LIN {X 0,Y 347.191,Z 710.482,A -85,B 0,C 180,E1 -13656.751,E2 -13656.751} C_VEL
LIN {X 0,Y 346.794,Z 715.502,A -85,B 0,C 180,E1 -13658.78,E2 -13658.78} C_VEL
LIN {X 0,Y 346.624,Z 717.5,A -85,B 0,C 180,E1 -13659.837,E2 -13659.837} C_VEL
LIN {X 0,Y 346.502,Z 719.364,A -85,B 0,C 180,E1 -13661.063,E2 -13661.063} C_VEL
LIN {X 0,Y 346.447,Z 720.875,A -85,B 0,C 180,E1 -13662.443,E2 -13662.443} C_VEL
LIN {X 0,Y 346.474,Z 722.066,A -85,B 0,C 180,E1 -13664.71,E2 -13664.71} C_VEL
LIN {X 0,Y 346.685,Z 721.819,A -85,B 0,C 180,E1 -13666.664,E2 -13666.664} C_VEL
LIN {X 0,Y 346.881,Z 720.668,A -85,B 0,C 180,E1 -13668.31,E2 -13668.31} C_VEL
LIN {X 0,Y 347.167,Z 719.319,A -85,B 0,C 180,E1 -13669.502,E2 -13669.502} C_VEL
LIN {X 0,Y 347.704,Z 716.397,A -85,B 0,C 180,E1 -13671.281,E2 -13671.281} C_VEL
LIN {X 0,Y 348.352,Z 712.378,A -85,B 0,C 180,E1 -13673.047,E2 -13673.047} C_VEL
LIN {X 0,Y 349.156,Z 707.164,A -85,B 0,C 180,E1 -13674.803,E2 -13674.803} C_VEL
LIN {X 0,Y 350.157,Z 700.612,A -85,B 0,C 180,E1 -13676.548,E2 -13676.548} C_VEL
LIN {X 0,Y 351.356,Z 692.175,A -85,B 0,C 180,E1 -13678.338,E2 -13678.338} C_VEL
LIN {X 0,Y 352.806,Z 682.143,A -85,B 0,C 180,E1 -13680,E2 -13680} C_VEL
LIN {X 0,Y 353.932,Z 672.637,A -85,B 0,C 180,E1 -13681.28,E2 -13681.28} C_VEL
LIN {X 0,Y 355.119,Z 662.198,A -85,B 0,C 180,E1 -13682.41,E2 -13682.41} C_VEL
LIN {X 0,Y 356.252,Z 650.75,A -85,B 0,C 180,E1 -13683.393,E2 -13683.393} C_VEL
LIN {X 0,Y 357.17,Z 638.174,A -85,B 0,C 180,E1 -13684.231,E2 -13684.231} C_VEL
LIN {X 0,Y 357.806,Z 624.931,A -85,B 0,C 180,E1 -13684.859,E2 -13684.859} C_VEL
LIN {X 0,Y 358.604,Z 602.211,A -85,B 0,C 180,E1 -13685.518,E2 -13685.518} C_VEL
LIN {X 0,Y 361.1,Z 543.407,A -85,B 0,C 180,E1 -13687.11,E2 -13687.11} C_VEL
LIN {X 0,Y 355.905,Z 531.692,A -85,B 0,C 180,E1 -13688.046,E2 -13688.046} C_VEL
LIN {X 0,Y 350.304,Z 521.591,A -85,B 0,C 180,E1 -13689.037,E2 -13689.037} C_VEL
LIN {X 0,Y 348.516,Z 518.327,A -85,B 0,C 180,E1 -13689.402,E2 -13689.402} C_VEL
LIN {X 0,Y 347.926,Z 516.149,A -85,B 0,C 180,E1 -13690.474,E2 -13690.474} C_VEL
LIN {X 0,Y 347.891,Z 516.152,A -85,B 0,C 180,E1 -13694.15,E2 -13694.15} C_VEL
LIN {X 0,Y 347.883,Z 516.149,A -85,B 0,C 180,E1 -13698.29,E2 -13698.29} C_VEL
LIN {X 0,Y 347.781,Z 516.162,A -85,B 0,C 180,E1 -13701.635,E2 -13701.635} C_VEL
LIN {X 0,Y 347.805,Z 516.16,A -85,B 0,C 180,E1 -13705.109,E2 -13705.109} C_VEL
LIN {X 0,Y 347.806,Z 516.155,A -85,B 0,C 180,E1 -13707.694,E2 -13707.694} C_VEL
LIN {X 0,Y 347.758,Z 516.161,A -85,B 0,C 180,E1 -13710.347,E2 -13710.347} C_VEL
LIN {X 0,Y 347.739,Z 516.164,A -85,B 0,C 180,E1 -13714.464,E2 -13714.464} C_VEL
LIN {X 0,Y 347.769,Z 516.162,A -85,B 0,C 180,E1 -13717.989,E2 -13717.989} C_VEL
LIN {X 0,Y 347.746,Z 516.166,A -85,B 0,C 180,E1 -13721.831,E2 -13721.831} C_VEL
LIN {X 0,Y 347.762,Z 516.169,A -85,B 0,C 180,E1 -13725.017,E2 -13725.017} C_VEL
LIN {X 0,Y 347.747,Z 516.172,A -85,B 0,C 180,E1 -13728.398,E2 -13728.398} C_VEL
LIN {X 0,Y 347.774,Z 516.166,A -85,B 0,C 180,E1 -13732.011,E2 -13732.011} C_VEL
LIN {X 0,Y 347.795,Z 516.377,A -85,B 0,C 180,E1 -13733.619,E2 -13733.619} C_VEL
LIN {X 0,Y 350.137,Z 524.59,A -85,B 0,C 180,E1 -13736.498,E2 -13736.498} C_VEL
LIN {X 0,Y 352.428,Z 533.84,A -85,B 0,C 180,E1 -13739.377,E2 -13739.377} C_VEL
LIN {X 0,Y 354.131,Z 542.797,A -85,B 0,C 180,E1 -13741.88,E2 -13741.88} C_VEL
LIN {X 0,Y 354.087,Z 545.377,A -85,B 0,C 180,E1 -13742.519,E2 -13742.519} C_VEL
LIN {X 0,Y 352.488,Z 556.664,A -85,B 0,C 180,E1 -13745.091,E2 -13745.091} C_VEL
LIN {X 0,Y 356.46,Z 577.198,A -85,B 0,C 180,E1 -13746.185,E2 -13746.185} C_VEL
LIN {X 0,Y 358.79,Z 595.546,A -85,B 0,C 180,E1 -13746.986,E2 -13746.986} C_VEL
LIN {X 0,Y 359.351,Z 604.886,A -85,B 0,C 180,E1 -13747.328,E2 -13747.328} C_VEL
LIN {X 0,Y 356.822,Z 668.886,A -85,B 0,C 180,E1 -13749.047,E2 -13749.047} C_VEL
LIN {X 0,Y 355.901,Z 682.744,A -85,B 0,C 180,E1 -13749.633,E2 -13749.633} C_VEL
LIN {X 0,Y 354.708,Z 694.487,A -85,B 0,C 180,E1 -13750.317,E2 -13750.317} C_VEL
LIN {X 0,Y 353.285,Z 706.996,A -85,B 0,C 180,E1 -13751.29,E2 -13751.29} C_VEL
LIN {X 0,Y 351.842,Z 718.372,A -85,B 0,C 180,E1 -13752.415,E2 -13752.415} C_VEL
LIN {X 0,Y 350.371,Z 732.515,A -85,B 0,C 180,E1 -13753.991,E2 -13753.991} C_VEL
LIN {X 0,Y 349.307,Z 742.889,A -85,B 0,C 180,E1 -13755.434,E2 -13755.434} C_VEL
LIN {X 0,Y 348.389,Z 751.27,A -85,B 0,C 180,E1 -13756.883,E2 -13756.883} C_VEL
LIN {X 0,Y 347.452,Z 759.439,A -85,B 0,C 180,E1 -13758.626,E2 -13758.626} C_VEL
LIN {X 0,Y 346.971,Z 764.991,A -85,B 0,C 180,E1 -13760.086,E2 -13760.086} C_VEL
LIN {X 0,Y 346.551,Z 770.397,A -85,B 0,C 180,E1 -13761.839,E2 -13761.839} C_VEL
LIN {X 0,Y 346.304,Z 774.601,A -85,B 0,C 180,E1 -13763.592,E2 -13763.592} C_VEL
LIN {X 0,Y 346.222,Z 777.723,A -85,B 0,C 180,E1 -13765.343,E2 -13765.343} C_VEL
LIN {X 0,Y 346.186,Z 779.27,A -85,B 0,C 180,E1 -13766.508,E2 -13766.508} C_VEL
LIN {X 0,Y 346.144,Z 780.358,A -85,B 0,C 180,E1 -13767.673,E2 -13767.673} C_VEL
LIN {X 0,Y 346.153,Z 781.038,A -85,B 0,C 180,E1 -13768.837,E2 -13768.837} C_VEL
LIN {X 0,Y 346.173,Z 781.328,A -85,B 0,C 180,E1 -13770,E2 -13770} C_VEL
LIN {X 0,Y 346.137,Z 781.219,A -85,B 0,C 180,E1 -13771.163,E2 -13771.163} C_VEL
LIN {X 0,Y 346.143,Z 780.669,A -85,B 0,C 180,E1 -13772.327,E2 -13772.327} C_VEL
LIN {X 0,Y 346.187,Z 779.723,A -85,B 0,C 180,E1 -13773.492,E2 -13773.492} C_VEL
LIN {X 0,Y 346.224,Z 778.38,A -85,B 0,C 180,E1 -13774.657,E2 -13774.657} C_VEL
LIN {X 0,Y 346.279,Z 776.247,A -85,B 0,C 180,E1 -13776.015,E2 -13776.015} C_VEL
LIN {X 0,Y 346.574,Z 771.638,A -85,B 0,C 180,E1 -13778.16,E2 -13778.16} C_VEL
LIN {X 0,Y 347.014,Z 766.599,A -85,B 0,C 180,E1 -13779.913,E2 -13779.913} C_VEL
LIN {X 0,Y 347.657,Z 760.231,A -85,B 0,C 180,E1 -13781.663,E2 -13781.663} C_VEL
LIN {X 0,Y 348.697,Z 752.269,A -85,B 0,C 180,E1 -13783.402,E2 -13783.402} C_VEL
LIN {X 0,Y 349.658,Z 744.139,A -85,B 0,C 180,E1 -13784.848,E2 -13784.848} C_VEL
LIN {X 0,Y 350.803,Z 734.199,A -85,B 0,C 180,E1 -13786.288,E2 -13786.288} C_VEL
LIN {X 0,Y 352.096,Z 722.923,A -85,B 0,C 180,E1 -13787.571,E2 -13787.571} C_VEL
LIN {X 0,Y 353.243,Z 711.857,A -85,B 0,C 180,E1 -13788.562,E2 -13788.562} C_VEL
LIN {X 0,Y 354.174,Z 700.659,A -85,B 0,C 180,E1 -13789.337,E2 -13789.337} C_VEL
LIN {X 0,Y 355.064,Z 687.97,A -85,B 0,C 180,E1 -13789.964,E2 -13789.964} C_VEL
LIN {X 0,Y 355.672,Z 674.624,A -85,B 0,C 180,E1 -13790.381,E2 -13790.381} C_VEL
LIN {X 0,Y 356.823,Z 601.554,A -85,B 0,C 180,E1 -13791.864,E2 -13791.864} C_VEL
LIN {X 0,Y 352.399,Z 568.881,A -85,B 0,C 180,E1 -13792.872,E2 -13792.872} C_VEL
LIN {X 0,Y 351.1,Z 560.278,A -85,B 0,C 180,E1 -13793.162,E2 -13793.162} C_VEL
LIN {X 0,Y 350.704,Z 555.734,A -85,B 0,C 180,E1 -13793.503,E2 -13793.503} C_VEL
LIN {X 0,Y 352.352,Z 539.207,A -85,B 0,C 180,E1 -13796.985,E2 -13796.985} C_VEL
LIN {X 0,Y 351.415,Z 533.126,A -85,B 0,C 180,E1 -13798.362,E2 -13798.362} C_VEL
LIN {X 0,Y 348.104,Z 517.735,A -85,B 0,C 180,E1 -13802.01,E2 -13802.01} C_VEL
LIN {X 0,Y 347.769,Z 516.167,A -85,B 0,C 180,E1 -13802.426,E2 -13802.426} C_VEL
LIN {X 0,Y 347.768,Z 516.16,A -85,B 0,C 180,E1 -13806.064,E2 -13806.064} C_VEL
LIN {X 0,Y 347.749,Z 516.137,A -85,B 0,C 180,E1 -13808.792,E2 -13808.792} C_VEL
LIN {X 0,Y 347.748,Z 516.169,A -85,B 0,C 180,E1 -13811.829,E2 -13811.829} C_VEL
LIN {X 0,Y 347.765,Z 516.164,A -85,B 0,C 180,E1 -13815.016,E2 -13815.016} C_VEL
LIN {X 0,Y 347.763,Z 516.155,A -85,B 0,C 180,E1 -13818.393,E2 -13818.393} C_VEL
LIN {X 0,Y 347.774,Z 516.16,A -85,B 0,C 180,E1 -13822.01,E2 -13822.01} C_VEL
LIN {X 0,Y 347.739,Z 516.17,A -85,B 0,C 180,E1 -13825.536,E2 -13825.536} C_VEL
LIN {X 0,Y 347.758,Z 516.152,A -85,B 0,C 180,E1 -13829.653,E2 -13829.653} C_VEL
LIN {X 0,Y 347.846,Z 516.155,A -85,B 0,C 180,E1 -13832.744,E2 -13832.744} C_VEL
LIN {X 0,Y 347.777,Z 516.142,A -85,B 0,C 180,E1 -13836.161,E2 -13836.161} C_VEL
LIN {X 0,Y 347.799,Z 516.159,A -85,B 0,C 180,E1 -13839.909,E2 -13839.909} C_VEL
LIN {X 0,Y 347.858,Z 516.14,A -85,B 0,C 180,E1 -13842.359,E2 -13842.359} C_VEL
LIN {X 0,Y 347.89,Z 516.145,A -85,B 0,C 180,E1 -13845.971,E2 -13845.971} C_VEL
LIN {X 0,Y 347.925,Z 516.136,A -85,B 0,C 180,E1 -13849.526,E2 -13849.526} C_VEL
LIN {X 0,Y 348.09,Z 516.108,A -85,B 0,C 180,E1 -13853.042,E2 -13853.042} C_VEL
LIN {X 0,Y 348.201,Z 516.103,A -85,B 0,C 180,E1 -13857.687,E2 -13857.687} C_VEL
LIN {X 0,Y 348.34,Z 516.066,A -85,B 0,C 180,E1 -13860,E2 -13860} C_VEL
LIN {X 0,Y 348.201,Z 516.103,A -85,B 0,C 180,E1 -13862.314,E2 -13862.314} C_VEL
LIN {X 0,Y 348.087,Z 516.11,A -85,B 0,C 180,E1 -13866.958,E2 -13866.958} C_VEL
LIN {X 0,Y 347.921,Z 516.137,A -85,B 0,C 180,E1 -13870.475,E2 -13870.475} C_VEL
LIN {X 0,Y 347.892,Z 516.144,A -85,B 0,C 180,E1 -13874.15,E2 -13874.15} C_VEL
LIN {X 0,Y 347.884,Z 516.144,A -85,B 0,C 180,E1 -13878.291,E2 -13878.291} C_VEL
LIN {X 0,Y 347.782,Z 516.155,A -85,B 0,C 180,E1 -13881.636,E2 -13881.636} C_VEL
LIN {X 0,Y 347.807,Z 516.155,A -85,B 0,C 180,E1 -13885.109,E2 -13885.109} C_VEL
LIN {X 0,Y 347.807,Z 516.156,A -85,B 0,C 180,E1 -13887.695,E2 -13887.695} C_VEL
LIN {X 0,Y 347.766,Z 516.154,A -85,B 0,C 180,E1 -13890.347,E2 -13890.347} C_VEL
LIN {X 0,Y 347.744,Z 516.162,A -85,B 0,C 180,E1 -13894.045,E2 -13894.045} C_VEL
LIN {X 0,Y 347.759,Z 516.17,A -85,B 0,C 180,E1 -13897.322,E2 -13897.322} C_VEL
LIN {X 0,Y 347.73,Z 516.167,A -85,B 0,C 180,E1 -13900.298,E2 -13900.298} C_VEL
LIN {X 0,Y 347.724,Z 516.168,A -85,B 0,C 180,E1 -13903.409,E2 -13903.409} C_VEL
LIN {X 0,Y 347.726,Z 516.169,A -85,B 0,C 180,E1 -13906.687,E2 -13906.687} C_VEL
LIN {X 0,Y 347.747,Z 516.166,A -85,B 0,C 180,E1 -13910.174,E2 -13910.174} C_VEL
LIN {X 0,Y 347.762,Z 516.166,A -85,B 0,C 180,E1 -13912.68,E2 -13912.68} C_VEL
LIN {X 0,Y 347.749,Z 516.164,A -85,B 0,C 180,E1 -13915.957,E2 -13915.957} C_VEL
LIN {X 0,Y 347.77,Z 516.166,A -85,B 0,C 180,E1 -13917.712,E2 -13917.712} C_VEL
LIN {X 0,Y 351.213,Z 530.188,A -85,B 0,C 180,E1 -13920.971,E2 -13920.971} C_VEL
LIN {X 0,Y 352.992,Z 539.619,A -85,B 0,C 180,E1 -13923.039,E2 -13923.039} C_VEL
LIN {X 0,Y 352.487,Z 549.164,A -85,B 0,C 180,E1 -13924.862,E2 -13924.862} C_VEL
LIN {X 0,Y 357.616,Z 575.434,A -85,B 0,C 180,E1 -13925.813,E2 -13925.813} C_VEL
LIN {X 0,Y 357.927,Z 578.608,A -85,B 0,C 180,E1 -13925.902,E2 -13925.902} C_VEL
LIN {X 0,Y 356.197,Z 660.018,A -85,B 0,C 180,E1 -13927.564,E2 -13927.564} C_VEL
LIN {X 0,Y 355.59,Z 672.934,A -85,B 0,C 180,E1 -13928.045,E2 -13928.045} C_VEL
LIN {X 0,Y 354.85,Z 685.894,A -85,B 0,C 180,E1 -13928.789,E2 -13928.789} C_VEL
LIN {X 0,Y 353.861,Z 697.311,A -85,B 0,C 180,E1 -13929.662,E2 -13929.662} C_VEL
LIN {X 0,Y 352.65,Z 708.811,A -85,B 0,C 180,E1 -13930.803,E2 -13930.803} C_VEL
LIN {X 0,Y 351.376,Z 719.111,A -85,B 0,C 180,E1 -13932.091,E2 -13932.091} C_VEL
LIN {X 0,Y 350.306,Z 727.549,A -85,B 0,C 180,E1 -13933.388,E2 -13933.388} C_VEL
LIN {X 0,Y 349.2,Z 736.245,A -85,B 0,C 180,E1 -13935.03,E2 -13935.03} C_VEL
LIN {X 0,Y 348.309,Z 743.998,A -85,B 0,C 180,E1 -13936.88,E2 -13936.88} C_VEL
LIN {X 0,Y 347.34,Z 750.728,A -85,B 0,C 180,E1 -13938.918,E2 -13938.918} C_VEL
LIN {X 0,Y 346.849,Z 755.133,A -85,B 0,C 180,E1 -13940.671,E2 -13940.671} C_VEL
LIN {X 0,Y 346.612,Z 757.443,A -85,B 0,C 180,E1 -13941.84,E2 -13941.84} C_VEL
LIN {X 0,Y 346.328,Z 760.492,A -85,B 0,C 180,E1 -13943.913,E2 -13943.913} C_VEL
LIN {X 0,Y 346.228,Z 761.819,A -85,B 0,C 180,E1 -13945.343,E2 -13945.343} C_VEL
LIN {X 0,Y 346.122,Z 762.712,A -85,B 0,C 180,E1 -13947.673,E2 -13947.673} C_VEL
LIN {X 0,Y 346.132,Z 762.561,A -85,B 0,C 180,E1 -13948.837,E2 -13948.837} C_VEL
LIN {X 0,Y 346.168,Z 761.996,A -85,B 0,C 180,E1 -13950,E2 -13950} C_VEL
LIN {X 0,Y 346.335,Z 759.716,A -85,B 0,C 180,E1 -13952.326,E2 -13952.326} C_VEL
LIN {X 0,Y 346.569,Z 756.887,A -85,B 0,C 180,E1 -13954.07,E2 -13954.07} C_VEL
LIN {X 0,Y 346.939,Z 753.039,A -85,B 0,C 180,E1 -13955.813,E2 -13955.813} C_VEL
LIN {X 0,Y 347.481,Z 747.696,A -85,B 0,C 180,E1 -13957.665,E2 -13957.665} C_VEL
LIN {X 0,Y 348.24,Z 740.577,A -85,B 0,C 180,E1 -13959.584,E2 -13959.584} C_VEL
LIN {X 0,Y 349.222,Z 732.487,A -85,B 0,C 180,E1 -13961.316,E2 -13961.316} C_VEL
LIN {X 0,Y 350.217,Z 724.154,A -85,B 0,C 180,E1 -13962.752,E2 -13962.752} C_VEL
LIN {X 0,Y 351.299,Z 713.922,A -85,B 0,C 180,E1 -13964.186,E2 -13964.186} C_VEL
LIN {X 0,Y 352.354,Z 703.817,A -85,B 0,C 180,E1 -13965.324,E2 -13965.324} C_VEL
LIN {X 0,Y 353.317,Z 692.746,A -85,B 0,C 180,E1 -13966.318,E2 -13966.318} C_VEL
LIN {X 0,Y 354.286,Z 680.233,A -85,B 0,C 180,E1 -13967.162,E2 -13967.162} C_VEL
LIN {X 0,Y 354.855,Z 667.182,A -85,B 0,C 180,E1 -13967.801,E2 -13967.801} C_VEL
LIN {X 0,Y 355.283,Z 653.229,A -85,B 0,C 180,E1 -13968.21,E2 -13968.21} C_VEL
LIN {X 0,Y 356.187,Z 606.958,A -85,B 0,C 180,E1 -13969.133,E2 -13969.133} C_VEL
LIN {X 0,Y 355.84,Z 601.151,A -85,B 0,C 180,E1 -13969.277,E2 -13969.277} C_VEL
LIN {X 0,Y 353.732,Z 591.744,A -85,B 0,C 180,E1 -13969.605,E2 -13969.605} C_VEL
LIN {X 0,Y 351.581,Z 584.287,A -85,B 0,C 180,E1 -13969.899,E2 -13969.899} C_VEL
LIN {X 0,Y 349.907,Z 576.693,A -85,B 0,C 180,E1 -13970.169,E2 -13970.169} C_VEL
LIN {X 0,Y 345.011,Z 549.363,A -85,B 0,C 180,E1 -13971.1,E2 -13971.1} C_VEL
LIN {X 0,Y 345.443,Z 539.348,A -85,B 0,C 180,E1 -13973.024,E2 -13973.024} C_VEL
LIN {X 0,Y 343.402,Z 528.311,A -85,B 0,C 180,E1 -13975.453,E2 -13975.453} C_VEL
LIN {X 0,Y 340.796,Z 517.036,A -85,B 0,C 180,E1 -13978.04,E2 -13978.04} C_VEL
LIN {X 0,Y 340.705,Z 517.046,A -85,B 0,C 180,E1 -13981.043,E2 -13981.043} C_VEL
LIN {X 0,Y 340.718,Z 517.044,A -85,B 0,C 180,E1 -13985.278,E2 -13985.278} C_VEL
LIN {X 0,Y 340.711,Z 517.045,A -85,B 0,C 180,E1 -13988.385,E2 -13988.385} C_VEL
LIN {X 0,Y 340.724,Z 517.039,A -85,B 0,C 180,E1 -13991.303,E2 -13991.303} C_VEL
LIN {X 0,Y 340.719,Z 517.034,A -85,B 0,C 180,E1 -13994.531,E2 -13994.531} C_VEL
LIN {X 0,Y 340.684,Z 517.05,A -85,B 0,C 180,E1 -13998.689,E2 -13998.689} C_VEL
LIN {X 0,Y 340.722,Z 517.043,A -85,B 0,C 180,E1 -14001.814,E2 -14001.814} C_VEL
LIN {X 0,Y 348.431,Z 538.596,A -85,B 0,C 180,E1 -14002.795,E2 -14002.795} C_VEL
LIN {X 0,Y 346.353,Z 619.657,A -85,B 0,C 180,E1 -14004.868,E2 -14004.868} C_VEL
LIN {X 0,Y 345.93,Z 632.4,A -85,B 0,C 180,E1 -14005.417,E2 -14005.417} C_VEL
LIN {X 0,Y 345.376,Z 644.462,A -85,B 0,C 180,E1 -14006.147,E2 -14006.147} C_VEL
LIN {X 0,Y 344.579,Z 656.447,A -85,B 0,C 180,E1 -14007.109,E2 -14007.109} C_VEL
LIN {X 0,Y 343.624,Z 668.932,A -85,B 0,C 180,E1 -14008.392,E2 -14008.392} C_VEL
LIN {X 0,Y 342.759,Z 679.979,A -85,B 0,C 180,E1 -14009.844,E2 -14009.844} C_VEL
LIN {X 0,Y 341.853,Z 689.836,A -85,B 0,C 180,E1 -14011.446,E2 -14011.446} C_VEL
LIN {X 0,Y 341.15,Z 697.81,A -85,B 0,C 180,E1 -14013.049,E2 -14013.049} C_VEL
LIN {X 0,Y 340.546,Z 705.253,A -85,B 0,C 180,E1 -14014.911,E2 -14014.911} C_VEL
LIN {X 0,Y 340.063,Z 711.466,A -85,B 0,C 180,E1 -14016.879,E2 -14016.879} C_VEL
LIN {X 0,Y 339.74,Z 715.579,A -85,B 0,C 180,E1 -14018.57,E2 -14018.57} C_VEL
LIN {X 0,Y 339.45,Z 719.287,A -85,B 0,C 180,E1 -14020.654,E2 -14020.654} C_VEL
LIN {X 0,Y 339.394,Z 721.231,A -85,B 0,C 180,E1 -14022.273,E2 -14022.273} C_VEL
LIN {X 0,Y 339.395,Z 722.535,A -85,B 0,C 180,E1 -14024.383,E2 -14024.383} C_VEL
LIN {X 0,Y 339.607,Z 722.495,A -85,B 0,C 180,E1 -14026.561,E2 -14026.561} C_VEL
LIN {X 0,Y 339.791,Z 721.654,A -85,B 0,C 180,E1 -14028.063,E2 -14028.063} C_VEL
LIN {X 0,Y 340.046,Z 720.452,A -85,B 0,C 180,E1 -14029.28,E2 -14029.28} C_VEL
LIN {X 0,Y 340.615,Z 717.8,A -85,B 0,C 180,E1 -14031.097,E2 -14031.097} C_VEL
LIN {X 0,Y 341.282,Z 714.089,A -85,B 0,C 180,E1 -14032.902,E2 -14032.902} C_VEL
LIN {X 0,Y 342.117,Z 709.218,A -85,B 0,C 180,E1 -14034.696,E2 -14034.696} C_VEL
LIN {X 0,Y 343.1,Z 703.059,A -85,B 0,C 180,E1 -14036.477,E2 -14036.477} C_VEL
LIN {X 0,Y 344.335,Z 695.007,A -85,B 0,C 180,E1 -14038.304,E2 -14038.304} C_VEL
LIN {X 0,Y 345.825,Z 685.582,A -85,B 0,C 180,E1 -14040,E2 -14040} C_VEL
LIN {X 0,Y 347.125,Z 675.585,A -85,B 0,C 180,E1 -14041.45,E2 -14041.45} C_VEL
LIN {X 0,Y 348.546,Z 664.355,A -85,B 0,C 180,E1 -14042.745,E2 -14042.745} C_VEL
LIN {X 0,Y 349.735,Z 653.39,A -85,B 0,C 180,E1 -14043.744,E2 -14043.744} C_VEL
LIN {X 0,Y 350.803,Z 640.159,A -85,B 0,C 180,E1 -14044.668,E2 -14044.668} C_VEL
LIN {X 0,Y 351.489,Z 627.703,A -85,B 0,C 180,E1 -14045.306,E2 -14045.306} C_VEL
LIN {X 0,Y 352.069,Z 611.332,A -85,B 0,C 180,E1 -14045.836,E2 -14045.836} C_VEL
LIN {X 0,Y 355.063,Z 545.537,A -85,B 0,C 180,E1 -14047.672,E2 -14047.672} C_VEL
LIN {X 0,Y 350.562,Z 535.405,A -85,B 0,C 180,E1 -14048.513,E2 -14048.513} C_VEL
LIN {X 0,Y 345.457,Z 526.088,A -85,B 0,C 180,E1 -14049.472,E2 -14049.472} C_VEL
LIN {X 0,Y 341.487,Z 519.336,A -85,B 0,C 180,E1 -14050.246,E2 -14050.246} C_VEL
LIN {X 0,Y 340.844,Z 517.03,A -85,B 0,C 180,E1 -14051.447,E2 -14051.447} C_VEL
LIN {X 0,Y 340.856,Z 517.029,A -85,B 0,C 180,E1 -14054.325,E2 -14054.325} C_VEL
LIN {X 0,Y 340.829,Z 517.028,A -85,B 0,C 180,E1 -14058.466,E2 -14058.466} C_VEL
LIN {X 0,Y 340.747,Z 517.038,A -85,B 0,C 180,E1 -14061.857,E2 -14061.857} C_VEL
LIN {X 0,Y 340.766,Z 517.033,A -85,B 0,C 180,E1 -14065.665,E2 -14065.665} C_VEL
LIN {X 0,Y 340.736,Z 517.036,A -85,B 0,C 180,E1 -14068.32,E2 -14068.32} C_VEL
LIN {X 0,Y 340.698,Z 517.043,A -85,B 0,C 180,E1 -14071.045,E2 -14071.045} C_VEL
LIN {X 0,Y 340.713,Z 517.042,A -85,B 0,C 180,E1 -14075.279,E2 -14075.279} C_VEL
LIN {X 0,Y 340.705,Z 517.042,A -85,B 0,C 180,E1 -14078.387,E2 -14078.387} C_VEL
LIN {X 0,Y 340.694,Z 517.044,A -85,B 0,C 180,E1 -14082.046,E2 -14082.046} C_VEL
LIN {X 0,Y 340.679,Z 517.049,A -85,B 0,C 180,E1 -14085.462,E2 -14085.462} C_VEL
LIN {X 0,Y 340.683,Z 517.05,A -85,B 0,C 180,E1 -14088.691,E2 -14088.691} C_VEL
LIN {X 0,Y 340.741,Z 517.155,A -85,B 0,C 180,E1 -14092.616,E2 -14092.616} C_VEL
LIN {X 0,Y 343.201,Z 525.658,A -85,B 0,C 180,E1 -14095.799,E2 -14095.799} C_VEL
LIN {X 0,Y 345.651,Z 535.486,A -85,B 0,C 180,E1 -14099.011,E2 -14099.011} C_VEL
LIN {X 0,Y 347.353,Z 544.47,A -85,B 0,C 180,E1 -14101.61,E2 -14101.61} C_VEL
LIN {X 0,Y 347.368,Z 547.045,A -85,B 0,C 180,E1 -14102.269,E2 -14102.269} C_VEL
LIN {X 0,Y 345.998,Z 555.843,A -85,B 0,C 180,E1 -14104.328,E2 -14104.328} C_VEL
LIN {X 0,Y 349.88,Z 575.095,A -85,B 0,C 180,E1 -14105.428,E2 -14105.428} C_VEL
LIN {X 0,Y 352.104,Z 591.203,A -85,B 0,C 180,E1 -14106.2,E2 -14106.2} C_VEL
LIN {X 0,Y 353.195,Z 604.961,A -85,B 0,C 180,E1 -14106.761,E2 -14106.761} C_VEL
LIN {X 0,Y 350.497,Z 669.155,A -85,B 0,C 180,E1 -14108.535,E2 -14108.535} C_VEL
LIN {X 0,Y 349.442,Z 683.271,A -85,B 0,C 180,E1 -14109.162,E2 -14109.162} C_VEL
LIN {X 0,Y 348.097,Z 695.544,A -85,B 0,C 180,E1 -14109.927,E2 -14109.927} C_VEL
LIN {X 0,Y 346.613,Z 707.641,A -85,B 0,C 180,E1 -14110.916,E2 -14110.916} C_VEL
LIN {X 0,Y 345.103,Z 718.738,A -85,B 0,C 180,E1 -14112.061,E2 -14112.061} C_VEL
LIN {X 0,Y 343.278,Z 734.494,A -85,B 0,C 180,E1 -14113.956,E2 -14113.956} C_VEL
LIN {X 0,Y 342.177,Z 744.421,A -85,B 0,C 180,E1 -14115.435,E2 -14115.435} C_VEL
LIN {X 0,Y 341.267,Z 752.483,A -85,B 0,C 180,E1 -14116.907,E2 -14116.907} C_VEL
LIN {X 0,Y 340.336,Z 760.405,A -85,B 0,C 180,E1 -14118.687,E2 -14118.687} C_VEL
LIN {X 0,Y 339.759,Z 766.704,A -85,B 0,C 180,E1 -14120.475,E2 -14120.475} C_VEL
LIN {X 0,Y 339.396,Z 771.695,A -85,B 0,C 180,E1 -14122.265,E2 -14122.265} C_VEL
LIN {X 0,Y 339.189,Z 775.535,A -85,B 0,C 180,E1 -14124.054,E2 -14124.054} C_VEL
LIN {X 0,Y 339.123,Z 777.506,A -85,B 0,C 180,E1 -14125.245,E2 -14125.245} C_VEL
LIN {X 0,Y 339.109,Z 779.059,A -85,B 0,C 180,E1 -14126.435,E2 -14126.435} C_VEL
LIN {X 0,Y 339.055,Z 780.156,A -85,B 0,C 180,E1 -14127.624,E2 -14127.624} C_VEL
LIN {X 0,Y 339.054,Z 780.84,A -85,B 0,C 180,E1 -14128.812,E2 -14128.812} C_VEL
LIN {X 0,Y 339.075,Z 781.135,A -85,B 0,C 180,E1 -14130,E2 -14130} C_VEL
LIN {X 0,Y 339.04,Z 781.033,A -85,B 0,C 180,E1 -14131.188,E2 -14131.188} C_VEL
LIN {X 0,Y 339.055,Z 780.49,A -85,B 0,C 180,E1 -14132.376,E2 -14132.376} C_VEL
LIN {X 0,Y 339.11,Z 779.549,A -85,B 0,C 180,E1 -14133.565,E2 -14133.565} C_VEL
LIN {X 0,Y 339.124,Z 778.209,A -85,B 0,C 180,E1 -14134.755,E2 -14134.755} C_VEL
LIN {X 0,Y 339.237,Z 775.369,A -85,B 0,C 180,E1 -14136.542,E2 -14136.542} C_VEL
LIN {X 0,Y 339.531,Z 771.489,A -85,B 0,C 180,E1 -14138.331,E2 -14138.331} C_VEL
LIN {X 0,Y 340.011,Z 766.462,A -85,B 0,C 180,E1 -14140.119,E2 -14140.119} C_VEL
LIN {X 0,Y 340.681,Z 760.114,A -85,B 0,C 180,E1 -14141.905,E2 -14141.905} C_VEL
LIN {X 0,Y 341.779,Z 752.168,A -85,B 0,C 180,E1 -14143.678,E2 -14143.678} C_VEL
LIN {X 0,Y 342.796,Z 744.057,A -85,B 0,C 180,E1 -14145.153,E2 -14145.153} C_VEL
LIN {X 0,Y 343.963,Z 734.146,A -85,B 0,C 180,E1 -14146.621,E2 -14146.621} C_VEL
LIN {X 0,Y 345.18,Z 724.323,A -85,B 0,C 180,E1 -14147.782,E2 -14147.782} C_VEL
LIN {X 0,Y 346.356,Z 713.636,A -85,B 0,C 180,E1 -14148.791,E2 -14148.791} C_VEL
LIN {X 0,Y 347.402,Z 701.87,A -85,B 0,C 180,E1 -14149.653,E2 -14149.653} C_VEL
LIN {X 0,Y 348.342,Z 689.138,A -85,B 0,C 180,E1 -14150.328,E2 -14150.328} C_VEL
LIN {X 0,Y 348.986,Z 676.648,A -85,B 0,C 180,E1 -14150.751,E2 -14150.751} C_VEL
LIN {X 0,Y 350.284,Z 602.378,A -85,B 0,C 180,E1 -14152.293,E2 -14152.293} C_VEL
LIN {X 0,Y 345.913,Z 569.839,A -85,B 0,C 180,E1 -14153.322,E2 -14153.322} C_VEL
LIN {X 0,Y 344.407,Z 560.047,A -85,B 0,C 180,E1 -14153.675,E2 -14153.675} C_VEL
LIN {X 0,Y 343.892,Z 554.129,A -85,B 0,C 180,E1 -14154.125,E2 -14154.125} C_VEL
LIN {X 0,Y 345.334,Z 541.093,A -85,B 0,C 180,E1 -14156.924,E2 -14156.924} C_VEL
LIN {X 0,Y 344.869,Z 536.598,A -85,B 0,C 180,E1 -14157.95,E2 -14157.95} C_VEL
LIN {X 0,Y 341.635,Z 521.206,A -85,B 0,C 180,E1 -14161.639,E2 -14161.639} C_VEL
LIN {X 0,Y 340.735,Z 517.044,A -85,B 0,C 180,E1 -14162.692,E2 -14162.692} C_VEL
LIN {X 0,Y 340.707,Z 517.03,A -85,B 0,C 180,E1 -14166.44,E2 -14166.44} C_VEL
LIN {X 0,Y 340.696,Z 517.029,A -85,B 0,C 180,E1 -14169.752,E2 -14169.752} C_VEL
LIN {X 0,Y 340.672,Z 517.046,A -85,B 0,C 180,E1 -14172.904,E2 -14172.904} C_VEL
LIN {X 0,Y 340.695,Z 517.047,A -85,B 0,C 180,E1 -14176.218,E2 -14176.218} C_VEL
LIN {X 0,Y 340.705,Z 517.045,A -85,B 0,C 180,E1 -14179.748,E2 -14179.748} C_VEL
LIN {X 0,Y 340.702,Z 517.034,A -85,B 0,C 180,E1 -14183.258,E2 -14183.258} C_VEL
LIN {X 0,Y 340.686,Z 517.046,A -85,B 0,C 180,E1 -14186.153,E2 -14186.153} C_VEL
LIN {X 0,Y 340.769,Z 517.025,A -85,B 0,C 180,E1 -14190.332,E2 -14190.332} C_VEL
LIN {X 0,Y 340.798,Z 517.035,A -85,B 0,C 180,E1 -14193.02,E2 -14193.02} C_VEL
LIN {X 0,Y 340.747,Z 517.018,A -85,B 0,C 180,E1 -14195.638,E2 -14195.638} C_VEL
LIN {X 0,Y 340.727,Z 517.042,A -85,B 0,C 180,E1 -14199.473,E2 -14199.473} C_VEL
LIN {X 0,Y 340.85,Z 517.014,A -85,B 0,C 180,E1 -14201.984,E2 -14201.984} C_VEL
LIN {X 0,Y 340.862,Z 517.022,A -85,B 0,C 180,E1 -14205.705,E2 -14205.705} C_VEL
LIN {X 0,Y 340.867,Z 517.017,A -85,B 0,C 180,E1 -14209.306,E2 -14209.306} C_VEL
LIN {X 0,Y 341.057,Z 516.982,A -85,B 0,C 180,E1 -14212.898,E2 -14212.898} C_VEL
LIN {X 0,Y 341.163,Z 516.98,A -85,B 0,C 180,E1 -14217.639,E2 -14217.639} C_VEL
LIN {X 0,Y 341.29,Z 516.943,A -85,B 0,C 180,E1 -14220,E2 -14220} C_VEL
LIN {X 0,Y 341.163,Z 516.979,A -85,B 0,C 180,E1 -14222.362,E2 -14222.362} C_VEL
LIN {X 0,Y 341.054,Z 516.984,A -85,B 0,C 180,E1 -14227.103,E2 -14227.103} C_VEL
LIN {X 0,Y 340.864,Z 517.017,A -85,B 0,C 180,E1 -14230.694,E2 -14230.694} C_VEL
LIN {X 0,Y 340.856,Z 517.021,A -85,B 0,C 180,E1 -14234.325,E2 -14234.325} C_VEL
LIN {X 0,Y 340.83,Z 517.023,A -85,B 0,C 180,E1 -14238.467,E2 -14238.467} C_VEL
LIN {X 0,Y 340.748,Z 517.031,A -85,B 0,C 180,E1 -14241.858,E2 -14241.858} C_VEL
LIN {X 0,Y 340.767,Z 517.036,A -85,B 0,C 180,E1 -14245.665,E2 -14245.665} C_VEL
LIN {X 0,Y 340.737,Z 517.036,A -85,B 0,C 180,E1 -14248.32,E2 -14248.32} C_VEL
LIN {X 0,Y 340.712,Z 517.039,A -85,B 0,C 180,E1 -14251.044,E2 -14251.044} C_VEL
LIN {X 0,Y 340.714,Z 517.036,A -85,B 0,C 180,E1 -14255.28,E2 -14255.28} C_VEL
LIN {X 0,Y 340.707,Z 517.047,A -85,B 0,C 180,E1 -14258.387,E2 -14258.387} C_VEL
LIN {X 0,Y 340.697,Z 517.049,A -85,B 0,C 180,E1 -14262.047,E2 -14262.047} C_VEL
LIN {X 0,Y 340.682,Z 517.05,A -85,B 0,C 180,E1 -14265.463,E2 -14265.463} C_VEL
LIN {X 0,Y 340.685,Z 517.05,A -85,B 0,C 180,E1 -14268.692,E2 -14268.692} C_VEL
LIN {X 0,Y 340.733,Z 517.038,A -85,B 0,C 180,E1 -14271.774,E2 -14271.774} C_VEL
LIN {X 0,Y 340.723,Z 517.035,A -85,B 0,C 180,E1 -14275.596,E2 -14275.596} C_VEL
LIN {X 0,Y 340.724,Z 517.085,A -85,B 0,C 180,E1 -14277.219,E2 -14277.219} C_VEL
LIN {X 0,Y 343.98,Z 530.104,A -85,B 0,C 180,E1 -14280.331,E2 -14280.331} C_VEL
LIN {X 0,Y 346.204,Z 541.28,A -85,B 0,C 180,E1 -14282.824,E2 -14282.824} C_VEL
LIN {X 0,Y 345.792,Z 549.609,A -85,B 0,C 180,E1 -14284.395,E2 -14284.395} C_VEL
LIN {X 0,Y 350.854,Z 575.149,A -85,B 0,C 180,E1 -14285.334,E2 -14285.334} C_VEL
LIN {X 0,Y 351.398,Z 579.233,A -85,B 0,C 180,E1 -14285.462,E2 -14285.462} C_VEL
LIN {X 0,Y 349.649,Z 659.3,A -85,B 0,C 180,E1 -14287.12,E2 -14287.12} C_VEL
LIN {X 0,Y 348.999,Z 672.794,A -85,B 0,C 180,E1 -14287.618,E2 -14287.618} C_VEL
LIN {X 0,Y 348.231,Z 685.556,A -85,B 0,C 180,E1 -14288.354,E2 -14288.354} C_VEL
LIN {X 0,Y 347.178,Z 697.213,A -85,B 0,C 180,E1 -14289.253,E2 -14289.253} C_VEL
LIN {X 0,Y 345.929,Z 708.791,A -85,B 0,C 180,E1 -14290.415,E2 -14290.415} C_VEL
LIN {X 0,Y 344.444,Z 720.168,A -85,B 0,C 180,E1 -14291.871,E2 -14291.871} C_VEL
LIN {X 0,Y 343.247,Z 729.298,A -85,B 0,C 180,E1 -14293.343,E2 -14293.343} C_VEL
LIN {X 0,Y 342.064,Z 738.14,A -85,B 0,C 180,E1 -14295.128,E2 -14295.128} C_VEL
LIN {X 0,Y 341.205,Z 745.193,A -85,B 0,C 180,E1 -14296.905,E2 -14296.905} C_VEL
LIN {X 0,Y 340.338,Z 750.852,A -85,B 0,C 180,E1 -14298.687,E2 -14298.687} C_VEL
LIN {X 0,Y 339.826,Z 755.274,A -85,B 0,C 180,E1 -14300.477,E2 -14300.477} C_VEL
LIN {X 0,Y 339.558,Z 757.592,A -85,B 0,C 180,E1 -14301.67,E2 -14301.67} C_VEL
LIN {X 0,Y 339.247,Z 760.831,A -85,B 0,C 180,E1 -14303.934,E2 -14303.934} C_VEL
LIN {X 0,Y 339.149,Z 761.994,A -85,B 0,C 180,E1 -14305.245,E2 -14305.245} C_VEL
LIN {X 0,Y 339.089,Z 762.636,A -85,B 0,C 180,E1 -14306.435,E2 -14306.435} C_VEL
LIN {X 0,Y 339.034,Z 762.9,A -85,B 0,C 180,E1 -14307.624,E2 -14307.624} C_VEL
LIN {X 0,Y 339.034,Z 762.762,A -85,B 0,C 180,E1 -14308.812,E2 -14308.812} C_VEL
LIN {X 0,Y 339.071,Z 762.202,A -85,B 0,C 180,E1 -14310,E2 -14310} C_VEL
LIN {X 0,Y 339.244,Z 759.935,A -85,B 0,C 180,E1 -14312.375,E2 -14312.375} C_VEL
LIN {X 0,Y 339.495,Z 757.119,A -85,B 0,C 180,E1 -14314.155,E2 -14314.155} C_VEL
LIN {X 0,Y 339.881,Z 753.284,A -85,B 0,C 180,E1 -14315.934,E2 -14315.934} C_VEL
LIN {X 0,Y 340.49,Z 747.453,A -85,B 0,C 180,E1 -14317.979,E2 -14317.979} C_VEL
LIN {X 0,Y 341.251,Z 740.86,A -85,B 0,C 180,E1 -14319.782,E2 -14319.782} C_VEL
LIN {X 0,Y 342.287,Z 732.791,A -85,B 0,C 180,E1 -14321.548,E2 -14321.548} C_VEL
LIN {X 0,Y 343.318,Z 724.488,A -85,B 0,C 180,E1 -14323.013,E2 -14323.013} C_VEL
LIN {X 0,Y 344.449,Z 714.282,A -85,B 0,C 180,E1 -14324.474,E2 -14324.474} C_VEL
LIN {X 0,Y 345.54,Z 704.211,A -85,B 0,C 180,E1 -14325.634,E2 -14325.634} C_VEL
LIN {X 0,Y 346.541,Z 693.205,A -85,B 0,C 180,E1 -14326.646,E2 -14326.646} C_VEL
LIN {X 0,Y 347.528,Z 680.778,A -85,B 0,C 180,E1 -14327.506,E2 -14327.506} C_VEL
LIN {X 0,Y 348.112,Z 668.093,A -85,B 0,C 180,E1 -14328.147,E2 -14328.147} C_VEL
LIN {X 0,Y 348.561,Z 654.621,A -85,B 0,C 180,E1 -14328.567,E2 -14328.567} C_VEL
LIN {X 0,Y 349.948,Z 576.965,A -85,B 0,C 180,E1 -14330.16,E2 -14330.16} C_VEL
LIN {X 0,Y 349.907,Z 576.693,A -85,B 0,C 180,E1 -14330.169,E2 -14330.169} C_VEL
LIN {X 0,Y 348.704,Z 573.037,A -85,B 0,C 180,E1 -14330.326,E2 -14330.326} C_VEL
LIN {X 0,Y 345.131,Z 567.751,A -85,B 0,C 180,E1 -14330.676,E2 -14330.676} C_VEL
LIN {X 0,Y 341.444,Z 562.504,A -85,B 0,C 180,E1 -14331.042,E2 -14331.042} C_VEL
LIN {X 0,Y 340.067,Z 558.89,A -85,B 0,C 180,E1 -14331.218,E2 -14331.218} C_VEL
LIN {X 0,Y 338.228,Z 549.527,A -85,B 0,C 180,E1 -14331.559,E2 -14331.559} C_VEL
LIN {X 0,Y 338.635,Z 540.949,A -85,B 0,C 180,E1 -14333.223,E2 -14333.223} C_VEL
LIN {X 0,Y 336.508,Z 529.712,A -85,B 0,C 180,E1 -14335.735,E2 -14335.735} C_VEL
LIN {X 0,Y 333.758,Z 517.913,A -85,B 0,C 180,E1 -14338.511,E2 -14338.511} C_VEL
LIN {X 0,Y 333.634,Z 517.929,A -85,B 0,C 180,E1 -14341.777,E2 -14341.777} C_VEL
LIN {X 0,Y 333.686,Z 517.92,A -85,B 0,C 180,E1 -14344.773,E2 -14344.773} C_VEL
LIN {X 0,Y 333.678,Z 517.922,A -85,B 0,C 180,E1 -14348.802,E2 -14348.802} C_VEL
LIN {X 0,Y 333.687,Z 517.92,A -85,B 0,C 180,E1 -14352.509,E2 -14352.509} C_VEL
LIN {X 0,Y 333.632,Z 517.916,A -85,B 0,C 180,E1 -14355.96,E2 -14355.96} C_VEL
LIN {X 0,Y 333.645,Z 517.925,A -85,B 0,C 180,E1 -14359.314,E2 -14359.314} C_VEL
LIN {X 0,Y 333.676,Z 517.922,A -85,B 0,C 180,E1 -14361.459,E2 -14361.459} C_VEL
LIN {X 0,Y 341.579,Z 540.099,A -85,B 0,C 180,E1 -14362.499,E2 -14362.499} C_VEL
LIN {X 0,Y 339.45,Z 620.15,A -85,B 0,C 180,E1 -14364.615,E2 -14364.615} C_VEL
LIN {X 0,Y 338.957,Z 634.061,A -85,B 0,C 180,E1 -14365.236,E2 -14365.236} C_VEL
LIN {X 0,Y 338.338,Z 646.332,A -85,B 0,C 180,E1 -14366.022,E2 -14366.022} C_VEL
LIN {X 0,Y 337.491,Z 658.633,A -85,B 0,C 180,E1 -14367.059,E2 -14367.059} C_VEL
LIN {X 0,Y 336.641,Z 669.245,A -85,B 0,C 180,E1 -14368.187,E2 -14368.187} C_VEL
LIN {X 0,Y 335.798,Z 679.738,A -85,B 0,C 180,E1 -14369.576,E2 -14369.576} C_VEL
LIN {X 0,Y 334.898,Z 689.333,A -85,B 0,C 180,E1 -14371.14,E2 -14371.14} C_VEL
LIN {X 0,Y 334.187,Z 697.547,A -85,B 0,C 180,E1 -14372.78,E2 -14372.78} C_VEL
LIN {X 0,Y 333.578,Z 704.465,A -85,B 0,C 180,E1 -14374.478,E2 -14374.478} C_VEL
LIN {X 0,Y 333.095,Z 710.602,A -85,B 0,C 180,E1 -14376.366,E2 -14376.366} C_VEL
LIN {X 0,Y 332.699,Z 715.604,A -85,B 0,C 180,E1 -14378.348,E2 -14378.348} C_VEL
LIN {X 0,Y 332.413,Z 719.122,A -85,B 0,C 180,E1 -14380.228,E2 -14380.228} C_VEL
LIN {X 0,Y 332.322,Z 721.539,A -85,B 0,C 180,E1 -14382.109,E2 -14382.109} C_VEL
LIN {X 0,Y 332.302,Z 722.944,A -85,B 0,C 180,E1 -14384.041,E2 -14384.041} C_VEL
LIN {X 0,Y 332.371,Z 723.288,A -85,B 0,C 180,E1 -14385.301,E2 -14385.301} C_VEL
LIN {X 0,Y 332.549,Z 723.143,A -85,B 0,C 180,E1 -14386.557,E2 -14386.557} C_VEL
LIN {X 0,Y 332.696,Z 722.587,A -85,B 0,C 180,E1 -14387.804,E2 -14387.804} C_VEL
LIN {X 0,Y 332.949,Z 721.593,A -85,B 0,C 180,E1 -14389.048,E2 -14389.048} C_VEL
LIN {X 0,Y 333.29,Z 720.104,A -85,B 0,C 180,E1 -14390.288,E2 -14390.288} C_VEL
LIN {X 0,Y 333.875,Z 717.307,A -85,B 0,C 180,E1 -14391.999,E2 -14391.999} C_VEL
LIN {X 0,Y 334.712,Z 712.853,A -85,B 0,C 180,E1 -14393.973,E2 -14393.973} C_VEL
LIN {X 0,Y 335.692,Z 707.452,A -85,B 0,C 180,E1 -14395.798,E2 -14395.798} C_VEL
LIN {X 0,Y 336.898,Z 700.686,A -85,B 0,C 180,E1 -14397.609,E2 -14397.609} C_VEL
LIN {X 0,Y 338.038,Z 693.717,A -85,B 0,C 180,E1 -14399.122,E2 -14399.122} C_VEL
LIN {X 0,Y 339.403,Z 685.421,A -85,B 0,C 180,E1 -14400.593,E2 -14400.593} C_VEL
LIN {X 0,Y 340.803,Z 675.22,A -85,B 0,C 180,E1 -14402.068,E2 -14402.068} C_VEL
LIN {X 0,Y 342.306,Z 663.738,A -85,B 0,C 180,E1 -14403.384,E2 -14403.384} C_VEL
LIN {X 0,Y 343.581,Z 652.345,A -85,B 0,C 180,E1 -14404.399,E2 -14404.399} C_VEL
LIN {X 0,Y 344.613,Z 639.994,A -85,B 0,C 180,E1 -14405.265,E2 -14405.265} C_VEL
LIN {X 0,Y 345.344,Z 627.265,A -85,B 0,C 180,E1 -14405.913,E2 -14405.913} C_VEL
LIN {X 0,Y 346.16,Z 608.114,A -85,B 0,C 180,E1 -14406.521,E2 -14406.521} C_VEL
LIN {X 0,Y 349.053,Z 547.672,A -85,B 0,C 180,E1 -14408.255,E2 -14408.255} C_VEL
LIN {X 0,Y 345.232,Z 539.034,A -85,B 0,C 180,E1 -14409.022,E2 -14409.022} C_VEL
LIN {X 0,Y 340.523,Z 530.408,A -85,B 0,C 180,E1 -14409.936,E2 -14409.936} C_VEL
LIN {X 0,Y 336.263,Z 523.502,A -85,B 0,C 180,E1 -14410.799,E2 -14410.799} C_VEL
LIN {X 0,Y 334.452,Z 520.265,A -85,B 0,C 180,E1 -14411.208,E2 -14411.208} C_VEL
LIN {X 0,Y 333.784,Z 517.908,A -85,B 0,C 180,E1 -14412.463,E2 -14412.463} C_VEL
LIN {X 0,Y 333.77,Z 517.911,A -85,B 0,C 180,E1 -14415.886,E2 -14415.886} C_VEL
LIN {X 0,Y 333.789,Z 517.906,A -85,B 0,C 180,E1 -14418.655,E2 -14418.655} C_VEL
LIN {X 0,Y 333.685,Z 517.919,A -85,B 0,C 180,E1 -14422.278,E2 -14422.278} C_VEL
LIN {X 0,Y 333.729,Z 517.911,A -85,B 0,C 180,E1 -14426.247,E2 -14426.247} C_VEL
LIN {X 0,Y 333.705,Z 517.914,A -85,B 0,C 180,E1 -14428.972,E2 -14428.972} C_VEL
LIN {X 0,Y 333.638,Z 517.921,A -85,B 0,C 180,E1 -14432.587,E2 -14432.587} C_VEL
LIN {X 0,Y 333.671,Z 517.916,A -85,B 0,C 180,E1 -14436.14,E2 -14436.14} C_VEL
LIN {X 0,Y 333.642,Z 517.927,A -85,B 0,C 180,E1 -14439.193,E2 -14439.193} C_VEL
LIN {X 0,Y 333.628,Z 517.926,A -85,B 0,C 180,E1 -14442.501,E2 -14442.501} C_VEL
LIN {X 0,Y 333.617,Z 517.929,A -85,B 0,C 180,E1 -14445.96,E2 -14445.96} C_VEL
LIN {X 0,Y 333.644,Z 517.927,A -85,B 0,C 180,E1 -14449.316,E2 -14449.316} C_VEL
LIN {X 0,Y 333.669,Z 518.007,A -85,B 0,C 180,E1 -14451.516,E2 -14451.516} C_VEL
LIN {X 0,Y 335.971,Z 525.722,A -85,B 0,C 180,E1 -14454.669,E2 -14454.669} C_VEL
LIN {X 0,Y 338.133,Z 534.074,A -85,B 0,C 180,E1 -14457.606,E2 -14457.606} C_VEL
LIN {X 0,Y 340.175,Z 543.502,A -85,B 0,C 180,E1 -14460.542,E2 -14460.542} C_VEL
LIN {X 0,Y 340.781,Z 547.49,A -85,B 0,C 180,E1 -14461.685,E2 -14461.685} C_VEL
LIN {X 0,Y 339.617,Z 555.073,A -85,B 0,C 180,E1 -14463.521,E2 -14463.521} C_VEL
LIN {X 0,Y 343.128,Z 572.133,A -85,B 0,C 180,E1 -14464.569,E2 -14464.569} C_VEL
LIN {X 0,Y 345.411,Z 586.562,A -85,B 0,C 180,E1 -14465.34,E2 -14465.34} C_VEL
LIN {X 0,Y 347.021,Z 603.168,A -85,B 0,C 180,E1 -14466.076,E2 -14466.076} C_VEL
LIN {X 0,Y 346.943,Z 609.244,A -85,B 0,C 180,E1 -14466.269,E2 -14466.269} C_VEL
LIN {X 0,Y 344.259,Z 668.434,A -85,B 0,C 180,E1 -14467.969,E2 -14467.969} C_VEL
LIN {X 0,Y 343.113,Z 682.555,A -85,B 0,C 180,E1 -14468.602,E2 -14468.602} C_VEL
LIN {X 0,Y 341.725,Z 694.829,A -85,B 0,C 180,E1 -14469.379,E2 -14469.379} C_VEL
LIN {X 0,Y 340.162,Z 706.941,A -85,B 0,C 180,E1 -14470.383,E2 -14470.383} C_VEL
LIN {X 0,Y 338.593,Z 718.011,A -85,B 0,C 180,E1 -14471.547,E2 -14471.547} C_VEL
LIN {X 0,Y 335.913,Z 738.418,A -85,B 0,C 180,E1 -14474.218,E2 -14474.218} C_VEL
LIN {X 0,Y 334.838,Z 747.532,A -85,B 0,C 180,E1 -14475.723,E2 -14475.723} C_VEL
LIN {X 0,Y 333.802,Z 756.399,A -85,B 0,C 180,E1 -14477.537,E2 -14477.537} C_VEL
LIN {X 0,Y 333.031,Z 763.486,A -85,B 0,C 180,E1 -14479.359,E2 -14479.359} C_VEL
LIN {X 0,Y 332.449,Z 769.923,A -85,B 0,C 180,E1 -14481.49,E2 -14481.49} C_VEL
LIN {X 0,Y 332.157,Z 774.147,A -85,B 0,C 180,E1 -14483.317,E2 -14483.317} C_VEL
LIN {X 0,Y 332.028,Z 777.289,A -85,B 0,C 180,E1 -14485.143,E2 -14485.143} C_VEL
LIN {X 0,Y 332.033,Z 778.848,A -85,B 0,C 180,E1 -14486.359,E2 -14486.359} C_VEL
LIN {X 0,Y 331.97,Z 779.954,A -85,B 0,C 180,E1 -14487.573,E2 -14487.573} C_VEL
LIN {X 0,Y 331.958,Z 780.642,A -85,B 0,C 180,E1 -14488.787,E2 -14488.787} C_VEL
LIN {X 0,Y 331.978,Z 780.942,A -85,B 0,C 180,E1 -14490,E2 -14490} C_VEL
LIN {X 0,Y 331.945,Z 780.846,A -85,B 0,C 180,E1 -14491.213,E2 -14491.213} C_VEL
LIN {X 0,Y 331.969,Z 780.311,A -85,B 0,C 180,E1 -14492.427,E2 -14492.427} C_VEL
LIN {X 0,Y 332.034,Z 779.374,A -85,B 0,C 180,E1 -14493.641,E2 -14493.641} C_VEL
LIN {X 0,Y 332.086,Z 776.529,A -85,B 0,C 180,E1 -14495.917,E2 -14495.917} C_VEL
LIN {X 0,Y 332.362,Z 772.764,A -85,B 0,C 180,E1 -14497.9,E2 -14497.9} C_VEL
LIN {X 0,Y 332.783,Z 768.135,A -85,B 0,C 180,E1 -14499.727,E2 -14499.727} C_VEL
LIN {X 0,Y 333.561,Z 761.13,A -85,B 0,C 180,E1 -14501.854,E2 -14501.854} C_VEL
LIN {X 0,Y 334.656,Z 753.54,A -85,B 0,C 180,E1 -14503.665,E2 -14503.665} C_VEL
LIN {X 0,Y 335.945,Z 743.977,A -85,B 0,C 180,E1 -14505.469,E2 -14505.469} C_VEL
LIN {X 0,Y 337.145,Z 734.092,A -85,B 0,C 180,E1 -14506.968,E2 -14506.968} C_VEL
LIN {X 0,Y 338.589,Z 722.9,A -85,B 0,C 180,E1 -14508.297,E2 -14508.297} C_VEL
LIN {X 0,Y 339.828,Z 711.925,A -85,B 0,C 180,E1 -14509.323,E2 -14509.323} C_VEL
LIN {X 0,Y 340.975,Z 699.715,A -85,B 0,C 180,E1 -14510.196,E2 -14510.196} C_VEL
LIN {X 0,Y 341.824,Z 686.75,A -85,B 0,C 180,E1 -14510.851,E2 -14510.851} C_VEL
LIN {X 0,Y 342.489,Z 674.346,A -85,B 0,C 180,E1 -14511.242,E2 -14511.242} C_VEL
LIN {X 0,Y 343.772,Z 603.154,A -85,B 0,C 180,E1 -14512.739,E2 -14512.739} C_VEL
LIN {X 0,Y 338.835,Z 566.34,A -85,B 0,C 180,E1 -14513.938,E2 -14513.938} C_VEL
LIN {X 0,Y 337.728,Z 559.865,A -85,B 0,C 180,E1 -14514.195,E2 -14514.195} C_VEL
LIN {X 0,Y 337.204,Z 552.373,A -85,B 0,C 180,E1 -14514.799,E2 -14514.799} C_VEL
LIN {X 0,Y 338.372,Z 541.515,A -85,B 0,C 180,E1 -14517.189,E2 -14517.189} C_VEL
LIN {X 0,Y 337.179,Z 534.256,A -85,B 0,C 180,E1 -14518.904,E2 -14518.904} C_VEL
LIN {X 0,Y 333.688,Z 517.922,A -85,B 0,C 180,E1 -14522.962,E2 -14522.962} C_VEL
LIN {X 0,Y 333.662,Z 517.899,A -85,B 0,C 180,E1 -14526.832,E2 -14526.832} C_VEL
LIN {X 0,Y 333.644,Z 517.921,A -85,B 0,C 180,E1 -14530.767,E2 -14530.767} C_VEL
LIN {X 0,Y 333.621,Z 517.921,A -85,B 0,C 180,E1 -14534.255,E2 -14534.255} C_VEL
LIN {X 0,Y 333.676,Z 517.911,A -85,B 0,C 180,E1 -14537.624,E2 -14537.624} C_VEL
LIN {X 0,Y 333.673,Z 517.922,A -85,B 0,C 180,E1 -14541.196,E2 -14541.196} C_VEL
LIN {X 0,Y 333.68,Z 517.918,A -85,B 0,C 180,E1 -14545.225,E2 -14545.225} C_VEL
LIN {X 0,Y 333.691,Z 517.903,A -85,B 0,C 180,E1 -14549.637,E2 -14549.637} C_VEL
LIN {X 0,Y 333.738,Z 517.911,A -85,B 0,C 180,E1 -14552.401,E2 -14552.401} C_VEL
LIN {X 0,Y 333.719,Z 517.897,A -85,B 0,C 180,E1 -14555.09,E2 -14555.09} C_VEL
LIN {X 0,Y 333.666,Z 517.92,A -85,B 0,C 180,E1 -14559.018,E2 -14559.018} C_VEL
LIN {X 0,Y 333.786,Z 517.896,A -85,B 0,C 180,E1 -14561.589,E2 -14561.589} C_VEL
LIN {X 0,Y 333.801,Z 517.898,A -85,B 0,C 180,E1 -14565.577,E2 -14565.577} C_VEL
LIN {X 0,Y 333.83,Z 517.896,A -85,B 0,C 180,E1 -14569.078,E2 -14569.078} C_VEL
LIN {X 0,Y 334.009,Z 517.858,A -85,B 0,C 180,E1 -14572.747,E2 -14572.747} C_VEL
LIN {X 0,Y 333.808,Z 517.905,A -85,B 0,C 180,E1 -14575.169,E2 -14575.169} C_VEL
LIN {X 0,Y 334.1,Z 517.86,A -85,B 0,C 180,E1 -14577.589,E2 -14577.589} C_VEL
LIN {X 0,Y 334.241,Z 517.821,A -85,B 0,C 180,E1 -14580,E2 -14580} C_VEL
LIN {X 0,Y 334.101,Z 517.859,A -85,B 0,C 180,E1 -14582.411,E2 -14582.411} C_VEL
LIN {X 0,Y 333.988,Z 517.867,A -85,B 0,C 180,E1 -14586.596,E2 -14586.596} C_VEL
LIN {X 0,Y 333.844,Z 517.885,A -85,B 0,C 180,E1 -14589.696,E2 -14589.696} C_VEL
LIN {X 0,Y 333.79,Z 517.903,A -85,B 0,C 180,E1 -14593.392,E2 -14593.392} C_VEL
LIN {X 0,Y 333.739,Z 517.894,A -85,B 0,C 180,E1 -14597.147,E2 -14597.147} C_VEL
LIN {X 0,Y 333.73,Z 517.913,A -85,B 0,C 180,E1 -14599.691,E2 -14599.691} C_VEL
LIN {X 0,Y 333.687,Z 517.909,A -85,B 0,C 180,E1 -14602.279,E2 -14602.279} C_VEL
LIN {X 0,Y 333.731,Z 517.912,A -85,B 0,C 180,E1 -14606.247,E2 -14606.247} C_VEL
LIN {X 0,Y 333.707,Z 517.904,A -85,B 0,C 180,E1 -14608.973,E2 -14608.973} C_VEL
LIN {X 0,Y 333.647,Z 517.925,A -85,B 0,C 180,E1 -14612.59,E2 -14612.59} C_VEL
LIN {X 0,Y 333.673,Z 517.919,A -85,B 0,C 180,E1 -14616.14,E2 -14616.14} C_VEL
LIN {X 0,Y 333.644,Z 517.92,A -85,B 0,C 180,E1 -14619.193,E2 -14619.193} C_VEL
LIN {X 0,Y 333.631,Z 517.93,A -85,B 0,C 180,E1 -14622.501,E2 -14622.501} C_VEL
LIN {X 0,Y 333.62,Z 517.928,A -85,B 0,C 180,E1 -14625.96,E2 -14625.96} C_VEL
LIN {X 0,Y 333.646,Z 517.921,A -85,B 0,C 180,E1 -14629.316,E2 -14629.316} C_VEL
LIN {X 0,Y 333.665,Z 517.925,A -85,B 0,C 180,E1 -14633.169,E2 -14633.169} C_VEL
LIN {X 0,Y 333.681,Z 517.991,A -85,B 0,C 180,E1 -14636.73,E2 -14636.73} C_VEL
LIN {X 0,Y 336.743,Z 529.983,A -85,B 0,C 180,E1 -14639.648,E2 -14639.648} C_VEL
LIN {X 0,Y 339.143,Z 541.185,A -85,B 0,C 180,E1 -14642.209,E2 -14642.209} C_VEL
LIN {X 0,Y 339.428,Z 544.555,A -85,B 0,C 180,E1 -14642.916,E2 -14642.916} C_VEL
LIN {X 0,Y 339.139,Z 549.814,A -85,B 0,C 180,E1 -14643.885,E2 -14643.885} C_VEL
LIN {X 0,Y 344.419,Z 576.436,A -85,B 0,C 180,E1 -14644.894,E2 -14644.894} C_VEL
LIN {X 0,Y 344.875,Z 580.444,A -85,B 0,C 180,E1 -14645.018,E2 -14645.018} C_VEL
LIN {X 0,Y 343.069,Z 659.892,A -85,B 0,C 180,E1 -14646.695,E2 -14646.695} C_VEL
LIN {X 0,Y 342.371,Z 673.222,A -85,B 0,C 180,E1 -14647.201,E2 -14647.201} C_VEL
LIN {X 0,Y 341.557,Z 686.37,A -85,B 0,C 180,E1 -14647.983,E2 -14647.983} C_VEL
LIN {X 0,Y 340.387,Z 698.777,A -85,B 0,C 180,E1 -14648.978,E2 -14648.978} C_VEL
LIN {X 0,Y 339.08,Z 710.023,A -85,B 0,C 180,E1 -14650.16,E2 -14650.16} C_VEL
LIN {X 0,Y 337.696,Z 720.186,A -85,B 0,C 180,E1 -14651.496,E2 -14651.496} C_VEL
LIN {X 0,Y 336.41,Z 729.357,A -85,B 0,C 180,E1 -14652.994,E2 -14652.994} C_VEL
LIN {X 0,Y 335.27,Z 737.456,A -85,B 0,C 180,E1 -14654.638,E2 -14654.638} C_VEL
LIN {X 0,Y 334.256,Z 745.295,A -85,B 0,C 180,E1 -14656.628,E2 -14656.628} C_VEL
LIN {X 0,Y 333.351,Z 750.976,A -85,B 0,C 180,E1 -14658.447,E2 -14658.447} C_VEL
LIN {X 0,Y 332.785,Z 755.415,A -85,B 0,C 180,E1 -14660.273,E2 -14660.273} C_VEL
LIN {X 0,Y 332.523,Z 757.741,A -85,B 0,C 180,E1 -14661.492,E2 -14661.492} C_VEL
LIN {X 0,Y 332.282,Z 759.643,A -85,B 0,C 180,E1 -14662.709,E2 -14662.709} C_VEL
LIN {X 0,Y 332.14,Z 761.203,A -85,B 0,C 180,E1 -14663.999,E2 -14663.999} C_VEL
LIN {X 0,Y 332.017,Z 762.818,A -85,B 0,C 180,E1 -14666.359,E2 -14666.359} C_VEL
LIN {X 0,Y 331.949,Z 763.087,A -85,B 0,C 180,E1 -14667.573,E2 -14667.573} C_VEL
LIN {X 0,Y 331.939,Z 762.961,A -85,B 0,C 180,E1 -14668.787,E2 -14668.787} C_VEL
LIN {X 0,Y 331.974,Z 762.409,A -85,B 0,C 180,E1 -14670,E2 -14670} C_VEL
LIN {X 0,Y 332.154,Z 760.155,A -85,B 0,C 180,E1 -14672.425,E2 -14672.425} C_VEL
LIN {X 0,Y 332.426,Z 757.35,A -85,B 0,C 180,E1 -14674.243,E2 -14674.243} C_VEL
LIN {X 0,Y 332.827,Z 753.529,A -85,B 0,C 180,E1 -14676.06,E2 -14676.06} C_VEL
LIN {X 0,Y 333.432,Z 747.963,A -85,B 0,C 180,E1 -14678.073,E2 -14678.073} C_VEL
LIN {X 0,Y 334.263,Z 741.143,A -85,B 0,C 180,E1 -14679.989,E2 -14679.989} C_VEL
LIN {X 0,Y 335.361,Z 733.092,A -85,B 0,C 180,E1 -14681.79,E2 -14681.79} C_VEL
LIN {X 0,Y 336.431,Z 724.82,A -85,B 0,C 180,E1 -14683.284,E2 -14683.284} C_VEL
LIN {X 0,Y 337.604,Z 714.641,A -85,B 0,C 180,E1 -14684.774,E2 -14684.774} C_VEL
LIN {X 0,Y 338.739,Z 704.603,A -85,B 0,C 180,E1 -14685.956,E2 -14685.956} C_VEL
LIN {X 0,Y 339.775,Z 693.654,A -85,B 0,C 180,E1 -14686.987,E2 -14686.987} C_VEL
LIN {X 0,Y 340.798,Z 681.32,A -85,B 0,C 180,E1 -14687.863,E2 -14687.863} C_VEL
LIN {X 0,Y 341.406,Z 668.582,A -85,B 0,C 180,E1 -14688.525,E2 -14688.525} C_VEL
LIN {X 0,Y 341.884,Z 655.907,A -85,B 0,C 180,E1 -14688.939,E2 -14688.939} C_VEL
LIN {X 0,Y 343.383,Z 578.072,A -85,B 0,C 180,E1 -14690.564,E2 -14690.564} C_VEL
LIN {X 0,Y 340.067,Z 558.89,A -85,B 0,C 180,E1 -14691.218,E2 -14691.218} C_VEL
LIN {X 0,Y 338.722,Z 555.273,A -85,B 0,C 180,E1 -14691.425,E2 -14691.425} C_VEL
LIN {X 0,Y 336.744,Z 552.17,A -85,B 0,C 180,E1 -14691.733,E2 -14691.733} C_VEL
LIN {X 0,Y 333.395,Z 547.706,A -85,B 0,C 180,E1 -14692.42,E2 -14692.42} C_VEL
LIN {X 0,Y 331.962,Z 544.7,A -85,B 0,C 180,E1 -14693.006,E2 -14693.006} C_VEL
LIN {X 0,Y 331.826,Z 543.387,A -85,B 0,C 180,E1 -14693.273,E2 -14693.273} C_VEL
LIN {X 0,Y 330.696,Z 536.16,A -85,B 0,C 180,E1 -14694.851,E2 -14694.851} C_VEL
LIN {X 0,Y 328.291,Z 525.22,A -85,B 0,C 180,E1 -14697.404,E2 -14697.404} C_VEL
LIN {X 0,Y 326.694,Z 518.791,A -85,B 0,C 180,E1 -14698.947,E2 -14698.947} C_VEL
LIN {X 0,Y 326.618,Z 518.8,A -85,B 0,C 180,E1 -14702.945,E2 -14702.945} C_VEL
LIN {X 0,Y 326.613,Z 518.8,A -85,B 0,C 180,E1 -14705.519,E2 -14705.519} C_VEL
LIN {X 0,Y 326.642,Z 518.793,A -85,B 0,C 180,E1 -14709.233,E2 -14709.233} C_VEL
LIN {X 0,Y 326.625,Z 518.8,A -85,B 0,C 180,E1 -14712.98,E2 -14712.98} C_VEL
LIN {X 0,Y 326.584,Z 518.802,A -85,B 0,C 180,E1 -14717.025,E2 -14717.025} C_VEL
LIN {X 0,Y 326.617,Z 518.807,A -85,B 0,C 180,E1 -14721.124,E2 -14721.124} C_VEL
LIN {X 0,Y 334.674,Z 541.446,A -85,B 0,C 180,E1 -14722.202,E2 -14722.202} C_VEL
LIN {X 0,Y 332.561,Z 620.658,A -85,B 0,C 180,E1 -14724.351,E2 -14724.351} C_VEL
LIN {X 0,Y 332.062,Z 634.129,A -85,B 0,C 180,E1 -14724.963,E2 -14724.963} C_VEL
LIN {X 0,Y 331.363,Z 647.081,A -85,B 0,C 180,E1 -14725.807,E2 -14725.807} C_VEL
LIN {X 0,Y 330.547,Z 658.707,A -85,B 0,C 180,E1 -14726.805,E2 -14726.805} C_VEL
LIN {X 0,Y 329.641,Z 670.123,A -85,B 0,C 180,E1 -14728.041,E2 -14728.041} C_VEL
LIN {X 0,Y 328.782,Z 680.747,A -85,B 0,C 180,E1 -14729.49,E2 -14729.49} C_VEL
LIN {X 0,Y 327.827,Z 690.374,A -85,B 0,C 180,E1 -14731.103,E2 -14731.103} C_VEL
LIN {X 0,Y 327.074,Z 698.734,A -85,B 0,C 180,E1 -14732.831,E2 -14732.831} C_VEL
LIN {X 0,Y 326.43,Z 706.058,A -85,B 0,C 180,E1 -14734.72,E2 -14734.72} C_VEL
LIN {X 0,Y 325.984,Z 711.58,A -85,B 0,C 180,E1 -14736.493,E2 -14736.493} C_VEL
LIN {X 0,Y 325.597,Z 716.396,A -85,B 0,C 180,E1 -14738.472,E2 -14738.472} C_VEL
LIN {X 0,Y 325.389,Z 718.885,A -85,B 0,C 180,E1 -14739.782,E2 -14739.782} C_VEL
LIN {X 0,Y 325.244,Z 721.832,A -85,B 0,C 180,E1 -14741.942,E2 -14741.942} C_VEL
LIN {X 0,Y 325.207,Z 723.27,A -85,B 0,C 180,E1 -14743.683,E2 -14743.683} C_VEL
LIN {X 0,Y 325.262,Z 723.781,A -85,B 0,C 180,E1 -14744.972,E2 -14744.972} C_VEL
LIN {X 0,Y 325.437,Z 723.854,A -85,B 0,C 180,E1 -14746.356,E2 -14746.356} C_VEL
LIN {X 0,Y 325.595,Z 723.465,A -85,B 0,C 180,E1 -14747.534,E2 -14747.534} C_VEL
LIN {X 0,Y 325.842,Z 722.621,A -85,B 0,C 180,E1 -14748.806,E2 -14748.806} C_VEL
LIN {X 0,Y 326.191,Z 721.352,A -85,B 0,C 180,E1 -14750.074,E2 -14750.074} C_VEL
LIN {X 0,Y 326.721,Z 719.034,A -85,B 0,C 180,E1 -14751.677,E2 -14751.677} C_VEL
LIN {X 0,Y 327.632,Z 714.691,A -85,B 0,C 180,E1 -14753.843,E2 -14753.843} C_VEL
LIN {X 0,Y 328.645,Z 709.646,A -85,B 0,C 180,E1 -14755.707,E2 -14755.707} C_VEL
LIN {X 0,Y 329.853,Z 703.249,A -85,B 0,C 180,E1 -14757.557,E2 -14757.557} C_VEL
LIN {X 0,Y 331.318,Z 695.114,A -85,B 0,C 180,E1 -14759.425,E2 -14759.425} C_VEL
LIN {X 0,Y 332.742,Z 687.085,A -85,B 0,C 180,E1 -14760.907,E2 -14760.907} C_VEL
LIN {X 0,Y 334.211,Z 677.152,A -85,B 0,C 180,E1 -14762.41,E2 -14762.41} C_VEL
LIN {X 0,Y 335.808,Z 666.043,A -85,B 0,C 180,E1 -14763.75,E2 -14763.75} C_VEL
LIN {X 0,Y 337.139,Z 655.265,A -85,B 0,C 180,E1 -14764.783,E2 -14764.783} C_VEL
LIN {X 0,Y 338.333,Z 642.358,A -85,B 0,C 180,E1 -14765.737,E2 -14765.737} C_VEL
LIN {X 0,Y 339.182,Z 629.48,A -85,B 0,C 180,E1 -14766.439,E2 -14766.439} C_VEL
LIN {X 0,Y 339.873,Z 613.069,A -85,B 0,C 180,E1 -14767.006,E2 -14767.006} C_VEL
LIN {X 0,Y 343.187,Z 549.889,A -85,B 0,C 180,E1 -14768.873,E2 -14768.873} C_VEL
LIN {X 0,Y 339.344,Z 541.399,A -85,B 0,C 180,E1 -14769.669,E2 -14769.669} C_VEL
LIN {X 0,Y 334.242,Z 532.263,A -85,B 0,C 180,E1 -14770.733,E2 -14770.733} C_VEL
LIN {X 0,Y 329.226,Z 524.405,A -85,B 0,C 180,E1 -14771.808,E2 -14771.808} C_VEL
LIN {X 0,Y 327.418,Z 521.274,A -85,B 0,C 180,E1 -14772.253,E2 -14772.253} C_VEL
LIN {X 0,Y 326.753,Z 518.783,A -85,B 0,C 180,E1 -14773.685,E2 -14773.685} C_VEL
LIN {X 0,Y 326.692,Z 518.792,A -85,B 0,C 180,E1 -14777.528,E2 -14777.528} C_VEL
LIN {X 0,Y 326.655,Z 518.794,A -85,B 0,C 180,E1 -14780.135,E2 -14780.135} C_VEL
LIN {X 0,Y 326.645,Z 518.794,A -85,B 0,C 180,E1 -14784.129,E2 -14784.129} C_VEL
LIN {X 0,Y 326.679,Z 518.792,A -85,B 0,C 180,E1 -14786.858,E2 -14786.858} C_VEL
LIN {X 0,Y 326.633,Z 518.794,A -85,B 0,C 180,E1 -14790.612,E2 -14790.612} C_VEL
LIN {X 0,Y 326.601,Z 518.796,A -85,B 0,C 180,E1 -14794.02,E2 -14794.02} C_VEL
LIN {X 0,Y 326.623,Z 518.8,A -85,B 0,C 180,E1 -14797.239,E2 -14797.239} C_VEL
LIN {X 0,Y 326.574,Z 518.808,A -85,B 0,C 180,E1 -14801.132,E2 -14801.132} C_VEL
LIN {X 0,Y 326.552,Z 518.811,A -85,B 0,C 180,E1 -14804.749,E2 -14804.749} C_VEL
LIN {X 0,Y 326.573,Z 518.81,A -85,B 0,C 180,E1 -14808.155,E2 -14808.155} C_VEL
LIN {X 0,Y 326.622,Z 518.972,A -85,B 0,C 180,E1 -14810.341,E2 -14810.341} C_VEL
LIN {X 0,Y 328.619,Z 525.347,A -85,B 0,C 180,E1 -14813.216,E2 -14813.216} C_VEL
LIN {X 0,Y 330.586,Z 532.578,A -85,B 0,C 180,E1 -14816.007,E2 -14816.007} C_VEL
LIN {X 0,Y 332.556,Z 540.807,A -85,B 0,C 180,E1 -14818.818,E2 -14818.818} C_VEL
LIN {X 0,Y 334.056,Z 549.388,A -85,B 0,C 180,E1 -14821.44,E2 -14821.44} C_VEL
LIN {X 0,Y 333.31,Z 554.259,A -85,B 0,C 180,E1 -14822.649,E2 -14822.649} C_VEL
LIN {X 0,Y 337.05,Z 572.032,A -85,B 0,C 180,E1 -14823.827,E2 -14823.827} C_VEL
LIN {X 0,Y 339.566,Z 588.246,A -85,B 0,C 180,E1 -14824.731,E2 -14824.731} C_VEL
LIN {X 0,Y 341.016,Z 604.534,A -85,B 0,C 180,E1 -14825.487,E2 -14825.487} C_VEL
LIN {X 0,Y 339.353,Z 643.2,A -85,B 0,C 180,E1 -14826.62,E2 -14826.62} C_VEL
LIN {X 0,Y 338.059,Z 668.381,A -85,B 0,C 180,E1 -14827.382,E2 -14827.382} C_VEL
LIN {X 0,Y 336.864,Z 682.106,A -85,B 0,C 180,E1 -14828.024,E2 -14828.024} C_VEL
LIN {X 0,Y 335.41,Z 694.218,A -85,B 0,C 180,E1 -14828.811,E2 -14828.811} C_VEL
LIN {X 0,Y 333.535,Z 707.791,A -85,B 0,C 180,E1 -14829.977,E2 -14829.977} C_VEL
LIN {X 0,Y 331.693,Z 719.728,A -85,B 0,C 180,E1 -14831.309,E2 -14831.309} C_VEL
LIN {X 0,Y 330.075,Z 729.493,A -85,B 0,C 180,E1 -14832.658,E2 -14832.658} C_VEL
LIN {X 0,Y 328.709,Z 741.838,A -85,B 0,C 180,E1 -14834.47,E2 -14834.47} C_VEL
LIN {X 0,Y 327.607,Z 750.451,A -85,B 0,C 180,E1 -14836.035,E2 -14836.035} C_VEL
LIN {X 0,Y 326.482,Z 758.658,A -85,B 0,C 180,E1 -14837.885,E2 -14837.885} C_VEL
LIN {X 0,Y 325.891,Z 764.246,A -85,B 0,C 180,E1 -14839.438,E2 -14839.438} C_VEL
LIN {X 0,Y 325.384,Z 769.685,A -85,B 0,C 180,E1 -14841.304,E2 -14841.304} C_VEL
LIN {X 0,Y 325.079,Z 773.92,A -85,B 0,C 180,E1 -14843.171,E2 -14843.171} C_VEL
LIN {X 0,Y 324.939,Z 777.072,A -85,B 0,C 180,E1 -14845.037,E2 -14845.037} C_VEL
LIN {X 0,Y 324.937,Z 778.636,A -85,B 0,C 180,E1 -14846.28,E2 -14846.28} C_VEL
LIN {X 0,Y 324.887,Z 779.752,A -85,B 0,C 180,E1 -14847.52,E2 -14847.52} C_VEL
LIN {X 0,Y 324.866,Z 780.444,A -85,B 0,C 180,E1 -14848.76,E2 -14848.76} C_VEL
LIN {X 0,Y 324.882,Z 780.748,A -85,B 0,C 180,E1 -14850,E2 -14850} C_VEL
LIN {X 0,Y 324.853,Z 780.659,A -85,B 0,C 180,E1 -14851.24,E2 -14851.24} C_VEL
LIN {X 0,Y 324.887,Z 780.132,A -85,B 0,C 180,E1 -14852.48,E2 -14852.48} C_VEL
LIN {X 0,Y 324.938,Z 779.199,A -85,B 0,C 180,E1 -14853.72,E2 -14853.72} C_VEL
LIN {X 0,Y 325.001,Z 776.599,A -85,B 0,C 180,E1 -14855.884,E2 -14855.884} C_VEL
LIN {X 0,Y 325.29,Z 772.615,A -85,B 0,C 180,E1 -14858.073,E2 -14858.073} C_VEL
LIN {X 0,Y 325.77,Z 767.998,A -85,B 0,C 180,E1 -14859.938,E2 -14859.938} C_VEL
LIN {X 0,Y 326.594,Z 761.007,A -85,B 0,C 180,E1 -14862.111,E2 -14862.111} C_VEL
LIN {X 0,Y 327.749,Z 753.436,A -85,B 0,C 180,E1 -14863.959,E2 -14863.959} C_VEL
LIN {X 0,Y 329.011,Z 744.461,A -85,B 0,C 180,E1 -14865.703,E2 -14865.703} C_VEL
LIN {X 0,Y 330.349,Z 734.037,A -85,B 0,C 180,E1 -14867.328,E2 -14867.328} C_VEL
LIN {X 0,Y 331.841,Z 722.891,A -85,B 0,C 180,E1 -14868.682,E2 -14868.682} C_VEL
LIN {X 0,Y 333.147,Z 711.961,A -85,B 0,C 180,E1 -14869.726,E2 -14869.726} C_VEL
LIN {X 0,Y 334.329,Z 699.838,A -85,B 0,C 180,E1 -14870.616,E2 -14870.616} C_VEL
LIN {X 0,Y 335.213,Z 687.034,A -85,B 0,C 180,E1 -14871.282,E2 -14871.282} C_VEL
LIN {X 0,Y 335.959,Z 673.495,A -85,B 0,C 180,E1 -14871.716,E2 -14871.716} C_VEL
LIN {X 0,Y 337.335,Z 604.683,A -85,B 0,C 180,E1 -14873.18,E2 -14873.18} C_VEL
LIN {X 0,Y 332.726,Z 569.527,A -85,B 0,C 180,E1 -14874.35,E2 -14874.35} C_VEL
LIN {X 0,Y 331.122,Z 560.076,A -85,B 0,C 180,E1 -14874.711,E2 -14874.711} C_VEL
LIN {X 0,Y 330.444,Z 550.743,A -85,B 0,C 180,E1 -14875.468,E2 -14875.468} C_VEL
LIN {X 0,Y 331.393,Z 542.48,A -85,B 0,C 180,E1 -14877.321,E2 -14877.321} C_VEL
LIN {X 0,Y 330.196,Z 535.582,A -85,B 0,C 180,E1 -14878.993,E2 -14878.993} C_VEL
LIN {X 0,Y 326.982,Z 520.455,A -85,B 0,C 180,E1 -14882.811,E2 -14882.811} C_VEL
LIN {X 0,Y 326.629,Z 518.801,A -85,B 0,C 180,E1 -14883.285,E2 -14883.285} C_VEL
LIN {X 0,Y 326.625,Z 518.769,A -85,B 0,C 180,E1 -14887.238,E2 -14887.238} C_VEL
LIN {X 0,Y 326.575,Z 518.805,A -85,B 0,C 180,E1 -14891.131,E2 -14891.131} C_VEL
LIN {X 0,Y 326.559,Z 518.803,A -85,B 0,C 180,E1 -14894.748,E2 -14894.748} C_VEL
LIN {X 0,Y 326.598,Z 518.791,A -85,B 0,C 180,E1 -14898.158,E2 -14898.158} C_VEL
LIN {X 0,Y 326.639,Z 518.796,A -85,B 0,C 180,E1 -14901.394,E2 -14901.394} C_VEL
LIN {X 0,Y 326.614,Z 518.794,A -85,B 0,C 180,E1 -14904.851,E2 -14904.851} C_VEL
LIN {X 0,Y 326.602,Z 518.796,A -85,B 0,C 180,E1 -14907.455,E2 -14907.455} C_VEL
LIN {X 0,Y 326.655,Z 518.783,A -85,B 0,C 180,E1 -14910.34,E2 -14910.34} C_VEL
LIN {X 0,Y 326.683,Z 518.782,A -85,B 0,C 180,E1 -14914.516,E2 -14914.516} C_VEL
LIN {X 0,Y 326.612,Z 518.795,A -85,B 0,C 180,E1 -14918.543,E2 -14918.543} C_VEL
LIN {X 0,Y 326.738,Z 518.777,A -85,B 0,C 180,E1 -14921.177,E2 -14921.177} C_VEL
LIN {X 0,Y 326.756,Z 518.773,A -85,B 0,C 180,E1 -14925.433,E2 -14925.433} C_VEL
LIN {X 0,Y 326.766,Z 518.779,A -85,B 0,C 180,E1 -14928.839,E2 -14928.839} C_VEL
LIN {X 0,Y 326.962,Z 518.734,A -85,B 0,C 180,E1 -14932.59,E2 -14932.59} C_VEL
LIN {X 0,Y 326.775,Z 518.779,A -85,B 0,C 180,E1 -14935.065,E2 -14935.065} C_VEL
LIN {X 0,Y 327.041,Z 518.739,A -85,B 0,C 180,E1 -14937.537,E2 -14937.537} C_VEL
LIN {X 0,Y 327.192,Z 518.698,A -85,B 0,C 180,E1 -14940,E2 -14940} C_VEL
LIN {X 0,Y 327.042,Z 518.739,A -85,B 0,C 180,E1 -14942.464,E2 -14942.464} C_VEL
LIN {X 0,Y 326.958,Z 518.744,A -85,B 0,C 180,E1 -14946.586,E2 -14946.586} C_VEL
LIN {X 0,Y 326.799,Z 518.765,A -85,B 0,C 180,E1 -14949.907,E2 -14949.907} C_VEL
LIN {X 0,Y 326.752,Z 518.778,A -85,B 0,C 180,E1 -14953.686,E2 -14953.686} C_VEL
LIN {X 0,Y 326.692,Z 518.777,A -85,B 0,C 180,E1 -14957.529,E2 -14957.529} C_VEL
LIN {X 0,Y 326.656,Z 518.794,A -85,B 0,C 180,E1 -14960.136,E2 -14960.136} C_VEL
LIN {X 0,Y 326.646,Z 518.782,A -85,B 0,C 180,E1 -14964.13,E2 -14964.13} C_VEL
LIN {X 0,Y 326.68,Z 518.794,A -85,B 0,C 180,E1 -14966.859,E2 -14966.859} C_VEL
LIN {X 0,Y 326.637,Z 518.787,A -85,B 0,C 180,E1 -14970.613,E2 -14970.613} C_VEL
LIN {X 0,Y 326.605,Z 518.795,A -85,B 0,C 180,E1 -14974.02,E2 -14974.02} C_VEL
LIN {X 0,Y 326.625,Z 518.804,A -85,B 0,C 180,E1 -14977.24,E2 -14977.24} C_VEL
LIN {X 0,Y 326.576,Z 518.809,A -85,B 0,C 180,E1 -14981.132,E2 -14981.132} C_VEL
LIN {X 0,Y 326.555,Z 518.809,A -85,B 0,C 180,E1 -14984.749,E2 -14984.749} C_VEL
LIN {X 0,Y 326.575,Z 518.805,A -85,B 0,C 180,E1 -14988.155,E2 -14988.155} C_VEL
LIN {X 0,Y 326.597,Z 518.801,A -85,B 0,C 180,E1 -14991.389,E2 -14991.389} C_VEL
LIN {X 0,Y 326.619,Z 518.789,A -85,B 0,C 180,E1 -14994.852,E2 -14994.852} C_VEL
LIN {X 0,Y 326.644,Z 518.933,A -85,B 0,C 180,E1 -14996.226,E2 -14996.226} C_VEL
LIN {X 0,Y 329.819,Z 531.177,A -85,B 0,C 180,E1 -14999.243,E2 -14999.243} C_VEL
LIN {X 0,Y 332.317,Z 542.764,A -85,B 0,C 180,E1 -15001.93,E2 -15001.93} C_VEL
LIN {X 0,Y 332.646,Z 546.752,A -85,B 0,C 180,E1 -15002.774,E2 -15002.774} C_VEL
LIN {X 0,Y 332.455,Z 549.628,A -85,B 0,C 180,E1 -15003.333,E2 -15003.333} C_VEL
LIN {X 0,Y 338.003,Z 577.835,A -85,B 0,C 180,E1 -15004.44,E2 -15004.44} C_VEL
LIN {X 0,Y 338.402,Z 581.198,A -85,B 0,C 180,E1 -15004.548,E2 -15004.548} C_VEL
LIN {X 0,Y 336.506,Z 660.489,A -85,B 0,C 180,E1 -15006.254,E2 -15006.254} C_VEL
LIN {X 0,Y 335.768,Z 673.762,A -85,B 0,C 180,E1 -15006.774,E2 -15006.774} C_VEL
LIN {X 0,Y 334.94,Z 686.197,A -85,B 0,C 180,E1 -15007.524,E2 -15007.524} C_VEL
LIN {X 0,Y 333.747,Z 698.703,A -85,B 0,C 180,E1 -15008.539,E2 -15008.539} C_VEL
LIN {X 0,Y 332.393,Z 710.006,A -85,B 0,C 180,E1 -15009.744,E2 -15009.744} C_VEL
LIN {X 0,Y 330.964,Z 720.205,A -85,B 0,C 180,E1 -15011.106,E2 -15011.106} C_VEL
LIN {X 0,Y 329.592,Z 729.414,A -85,B 0,C 180,E1 -15012.631,E2 -15012.631} C_VEL
LIN {X 0,Y 328.293,Z 738.111,A -85,B 0,C 180,E1 -15014.441,E2 -15014.441} C_VEL
LIN {X 0,Y 327.324,Z 745.397,A -85,B 0,C 180,E1 -15016.339,E2 -15016.339} C_VEL
LIN {X 0,Y 326.353,Z 751.099,A -85,B 0,C 180,E1 -15018.195,E2 -15018.195} C_VEL
LIN {X 0,Y 325.761,Z 755.556,A -85,B 0,C 180,E1 -15020.062,E2 -15020.062} C_VEL
LIN {X 0,Y 325.476,Z 757.891,A -85,B 0,C 180,E1 -15021.307,E2 -15021.307} C_VEL
LIN {X 0,Y 325.079,Z 761.297,A -85,B 0,C 180,E1 -15023.795,E2 -15023.795} C_VEL
LIN {X 0,Y 324.946,Z 762.999,A -85,B 0,C 180,E1 -15026.28,E2 -15026.28} C_VEL
LIN {X 0,Y 324.868,Z 763.275,A -85,B 0,C 180,E1 -15027.52,E2 -15027.52} C_VEL
LIN {X 0,Y 324.848,Z 763.16,A -85,B 0,C 180,E1 -15028.76,E2 -15028.76} C_VEL
LIN {X 0,Y 324.878,Z 762.615,A -85,B 0,C 180,E1 -15030,E2 -15030} C_VEL
LIN {X 0,Y 325.068,Z 760.373,A -85,B 0,C 180,E1 -15032.478,E2 -15032.478} C_VEL
LIN {X 0,Y 325.36,Z 757.581,A -85,B 0,C 180,E1 -15034.336,E2 -15034.336} C_VEL
LIN {X 0,Y 325.778,Z 753.774,A -85,B 0,C 180,E1 -15036.192,E2 -15036.192} C_VEL
LIN {X 0,Y 326.438,Z 747.987,A -85,B 0,C 180,E1 -15038.325,E2 -15038.325} C_VEL
LIN {X 0,Y 327.291,Z 741.425,A -85,B 0,C 180,E1 -15040.204,E2 -15040.204} C_VEL
LIN {X 0,Y 328.425,Z 733.393,A -85,B 0,C 180,E1 -15042.042,E2 -15042.042} C_VEL
LIN {X 0,Y 329.547,Z 725.15,A -85,B 0,C 180,E1 -15043.567,E2 -15043.567} C_VEL
LIN {X 0,Y 330.773,Z 714.999,A -85,B 0,C 180,E1 -15045.086,E2 -15045.086} C_VEL
LIN {X 0,Y 331.953,Z 704.994,A -85,B 0,C 180,E1 -15046.291,E2 -15046.291} C_VEL
LIN {X 0,Y 333.021,Z 694.094,A -85,B 0,C 180,E1 -15047.343,E2 -15047.343} C_VEL
LIN {X 0,Y 334.077,Z 681.861,A -85,B 0,C 180,E1 -15048.235,E2 -15048.235} C_VEL
LIN {X 0,Y 334.73,Z 668.983,A -85,B 0,C 180,E1 -15048.921,E2 -15048.921} C_VEL
LIN {X 0,Y 335.235,Z 655.889,A -85,B 0,C 180,E1 -15049.357,E2 -15049.357} C_VEL
LIN {X 0,Y 336.772,Z 578.803,A -85,B 0,C 180,E1 -15050.997,E2 -15050.997} C_VEL
LIN {X 0,Y 331.73,Z 550.917,A -85,B 0,C 180,E1 -15051.997,E2 -15051.997} C_VEL
LIN {X 0,Y 331.505,Z 549.646,A -85,B 0,C 180,E1 -15052.051,E2 -15052.051} C_VEL
LIN {X 0,Y 331.826,Z 543.387,A -85,B 0,C 180,E1 -15053.273,E2 -15053.273} C_VEL
LIN {X 0,Y 331.501,Z 540.963,A -85,B 0,C 180,E1 -15053.798,E2 -15053.798} C_VEL
LIN {X 0,Y 329.814,Z 537.741,A -85,B 0,C 180,E1 -15054.603,E2 -15054.603} C_VEL
LIN {X 0,Y 323.044,Z 530.247,A -85,B 0,C 180,E1 -15056.8,E2 -15056.8} C_VEL
LIN {X 0,Y 321.463,Z 526.909,A -85,B 0,C 180,E1 -15057.658,E2 -15057.658} C_VEL
LIN {X 0,Y 319.65,Z 519.67,A -85,B 0,C 180,E1 -15059.468,E2 -15059.468} C_VEL
LIN {X 0,Y 319.577,Z 519.674,A -85,B 0,C 180,E1 -15063.352,E2 -15063.352} C_VEL
LIN {X 0,Y 319.559,Z 519.674,A -85,B 0,C 180,E1 -15066.427,E2 -15066.427} C_VEL
LIN {X 0,Y 319.582,Z 519.67,A -85,B 0,C 180,E1 -15069.673,E2 -15069.673} C_VEL
LIN {X 0,Y 319.595,Z 519.672,A -85,B 0,C 180,E1 -15073.474,E2 -15073.474} C_VEL
LIN {X 0,Y 319.563,Z 519.676,A -85,B 0,C 180,E1 -15077.017,E2 -15077.017} C_VEL
LIN {X 0,Y 319.598,Z 519.815,A -85,B 0,C 180,E1 -15080.767,E2 -15080.767} C_VEL
LIN {X 0,Y 327.869,Z 543.089,A -85,B 0,C 180,E1 -15081.905,E2 -15081.905} C_VEL
LIN {X 0,Y 325.65,Z 621.088,A -85,B 0,C 180,E1 -15084.073,E2 -15084.073} C_VEL
LIN {X 0,Y 325.158,Z 634.393,A -85,B 0,C 180,E1 -15084.689,E2 -15084.689} C_VEL
LIN {X 0,Y 324.518,Z 646.344,A -85,B 0,C 180,E1 -15085.468,E2 -15085.468} C_VEL
LIN {X 0,Y 323.598,Z 658.916,A -85,B 0,C 180,E1 -15086.557,E2 -15086.557} C_VEL
LIN {X 0,Y 322.649,Z 670.759,A -85,B 0,C 180,E1 -15087.866,E2 -15087.866} C_VEL
LIN {X 0,Y 321.782,Z 681.066,A -85,B 0,C 180,E1 -15089.3,E2 -15089.3} C_VEL
LIN {X 0,Y 320.85,Z 690.102,A -85,B 0,C 180,E1 -15090.832,E2 -15090.832} C_VEL
LIN {X 0,Y 320.099,Z 698.383,A -85,B 0,C 180,E1 -15092.543,E2 -15092.543} C_VEL
LIN {X 0,Y 319.434,Z 705.752,A -85,B 0,C 180,E1 -15094.427,E2 -15094.427} C_VEL
LIN {X 0,Y 318.868,Z 712.494,A -85,B 0,C 180,E1 -15096.626,E2 -15096.626} C_VEL
LIN {X 0,Y 318.482,Z 717.242,A -85,B 0,C 180,E1 -15098.647,E2 -15098.647} C_VEL
LIN {X 0,Y 318.221,Z 720.703,A -85,B 0,C 180,E1 -15100.653,E2 -15100.653} C_VEL
LIN {X 0,Y 318.162,Z 722.337,A -85,B 0,C 180,E1 -15101.985,E2 -15101.985} C_VEL
LIN {X 0,Y 318.129,Z 723.519,A -85,B 0,C 180,E1 -15103.31,E2 -15103.31} C_VEL
LIN {X 0,Y 318.157,Z 724.246,A -85,B 0,C 180,E1 -15104.628,E2 -15104.628} C_VEL
LIN {X 0,Y 318.346,Z 724.465,A -85,B 0,C 180,E1 -15106.251,E2 -15106.251} C_VEL
LIN {X 0,Y 318.721,Z 723.632,A -85,B 0,C 180,E1 -15108.553,E2 -15108.553} C_VEL
LIN {X 0,Y 319.082,Z 722.508,A -85,B 0,C 180,E1 -15109.851,E2 -15109.851} C_VEL
LIN {X 0,Y 319.657,Z 720.262,A -85,B 0,C 180,E1 -15111.63,E2 -15111.63} C_VEL
LIN {X 0,Y 320.544,Z 716.448,A -85,B 0,C 180,E1 -15113.706,E2 -15113.706} C_VEL
LIN {X 0,Y 321.593,Z 711.723,A -85,B 0,C 180,E1 -15115.613,E2 -15115.613} C_VEL
LIN {X 0,Y 322.813,Z 705.724,A -85,B 0,C 180,E1 -15117.504,E2 -15117.504} C_VEL
LIN {X 0,Y 324.284,Z 698.12,A -85,B 0,C 180,E1 -15119.406,E2 -15119.406} C_VEL
LIN {X 0,Y 326.088,Z 688.825,A -85,B 0,C 180,E1 -15121.235,E2 -15121.235} C_VEL
LIN {X 0,Y 327.643,Z 679.23,A -85,B 0,C 180,E1 -15122.766,E2 -15122.766} C_VEL
LIN {X 0,Y 329.321,Z 668.397,A -85,B 0,C 180,E1 -15124.13,E2 -15124.13} C_VEL
LIN {X 0,Y 330.905,Z 656.343,A -85,B 0,C 180,E1 -15125.331,E2 -15125.331} C_VEL
LIN {X 0,Y 332.204,Z 643.304,A -85,B 0,C 180,E1 -15126.323,E2 -15126.323} C_VEL
LIN {X 0,Y 333.117,Z 630.79,A -85,B 0,C 180,E1 -15127.032,E2 -15127.032} C_VEL
LIN {X 0,Y 333.829,Z 615.526,A -85,B 0,C 180,E1 -15127.598,E2 -15127.598} C_VEL
LIN {X 0,Y 337.416,Z 552.445,A -85,B 0,C 180,E1 -15129.495,E2 -15129.495} C_VEL
LIN {X 0,Y 334.719,Z 546.224,A -85,B 0,C 180,E1 -15130.105,E2 -15130.105} C_VEL
LIN {X 0,Y 329.789,Z 537.181,A -85,B 0,C 180,E1 -15131.174,E2 -15131.174} C_VEL
LIN {X 0,Y 324.706,Z 529.047,A -85,B 0,C 180,E1 -15132.335,E2 -15132.335} C_VEL
LIN {X 0,Y 322.376,Z 525.581,A -85,B 0,C 180,E1 -15132.877,E2 -15132.877} C_VEL
LIN {X 0,Y 320.437,Z 522.333,A -85,B 0,C 180,E1 -15133.395,E2 -15133.395} C_VEL
LIN {X 0,Y 319.712,Z 519.66,A -85,B 0,C 180,E1 -15135.078,E2 -15135.078} C_VEL
LIN {X 0,Y 319.667,Z 519.667,A -85,B 0,C 180,E1 -15139.255,E2 -15139.255} C_VEL
LIN {X 0,Y 319.563,Z 519.677,A -85,B 0,C 180,E1 -15143.32,E2 -15143.32} C_VEL
LIN {X 0,Y 319.629,Z 519.666,A -85,B 0,C 180,E1 -15146.088,E2 -15146.088} C_VEL
LIN {X 0,Y 319.584,Z 519.673,A -85,B 0,C 180,E1 -15148.934,E2 -15148.934} C_VEL
LIN {X 0,Y 319.526,Z 519.676,A -85,B 0,C 180,E1 -15151.862,E2 -15151.862} C_VEL
LIN {X 0,Y 319.575,Z 519.673,A -85,B 0,C 180,E1 -15155.544,E2 -15155.544} C_VEL
LIN {X 0,Y 319.554,Z 519.679,A -85,B 0,C 180,E1 -15159.669,E2 -15159.669} C_VEL
LIN {X 0,Y 319.553,Z 519.68,A -85,B 0,C 180,E1 -15163.468,E2 -15163.468} C_VEL
LIN {X 0,Y 319.557,Z 519.681,A -85,B 0,C 180,E1 -15167.018,E2 -15167.018} C_VEL
LIN {X 0,Y 319.553,Z 519.788,A -85,B 0,C 180,E1 -15168.931,E2 -15168.931} C_VEL
LIN {X 0,Y 321.737,Z 526.613,A -85,B 0,C 180,E1 -15172.294,E2 -15172.294} C_VEL
LIN {X 0,Y 323.914,Z 534.497,A -85,B 0,C 180,E1 -15175.537,E2 -15175.537} C_VEL
LIN {X 0,Y 325.863,Z 542.833,A -85,B 0,C 180,E1 -15178.505,E2 -15178.505} C_VEL
LIN {X 0,Y 327.317,Z 551.068,A -85,B 0,C 180,E1 -15181.113,E2 -15181.113} C_VEL
LIN {X 0,Y 327.047,Z 553.299,A -85,B 0,C 180,E1 -15181.708,E2 -15181.708} C_VEL
LIN {X 0,Y 331.119,Z 572.194,A -85,B 0,C 180,E1 -15183.056,E2 -15183.056} C_VEL
LIN {X 0,Y 333.788,Z 589.875,A -85,B 0,C 180,E1 -15184.094,E2 -15184.094} C_VEL
LIN {X 0,Y 335.187,Z 606.528,A -85,B 0,C 180,E1 -15184.881,E2 -15184.881} C_VEL
LIN {X 0,Y 331.992,Z 667.42,A -85,B 0,C 180,E1 -15186.739,E2 -15186.739} C_VEL
LIN {X 0,Y 330.804,Z 680.57,A -85,B 0,C 180,E1 -15187.353,E2 -15187.353} C_VEL
LIN {X 0,Y 329.139,Z 693.855,A -85,B 0,C 180,E1 -15188.223,E2 -15188.223} C_VEL
LIN {X 0,Y 327.369,Z 705.819,A -85,B 0,C 180,E1 -15189.255,E2 -15189.255} C_VEL
LIN {X 0,Y 325.649,Z 716.774,A -85,B 0,C 180,E1 -15190.458,E2 -15190.458} C_VEL
LIN {X 0,Y 323.711,Z 727.843,A -85,B 0,C 180,E1 -15191.979,E2 -15191.979} C_VEL
LIN {X 0,Y 321.48,Z 744.119,A -85,B 0,C 180,E1 -15194.577,E2 -15194.577} C_VEL
LIN {X 0,Y 320.271,Z 753.142,A -85,B 0,C 180,E1 -15196.356,E2 -15196.356} C_VEL
LIN {X 0,Y 319.229,Z 760.767,A -85,B 0,C 180,E1 -15198.25,E2 -15198.25} C_VEL
LIN {X 0,Y 318.481,Z 767.788,A -85,B 0,C 180,E1 -15200.474,E2 -15200.474} C_VEL
LIN {X 0,Y 318.095,Z 772.426,A -85,B 0,C 180,E1 -15202.382,E2 -15202.382} C_VEL
LIN {X 0,Y 317.904,Z 775.736,A -85,B 0,C 180,E1 -15204.171,E2 -15204.171} C_VEL
LIN {X 0,Y 317.843,Z 778.424,A -85,B 0,C 180,E1 -15206.197,E2 -15206.197} C_VEL
LIN {X 0,Y 317.806,Z 779.549,A -85,B 0,C 180,E1 -15207.465,E2 -15207.465} C_VEL
LIN {X 0,Y 317.776,Z 780.247,A -85,B 0,C 180,E1 -15208.733,E2 -15208.733} C_VEL
LIN {X 0,Y 317.79,Z 780.555,A -85,B 0,C 180,E1 -15210,E2 -15210} C_VEL
LIN {X 0,Y 317.765,Z 780.472,A -85,B 0,C 180,E1 -15211.267,E2 -15211.267} C_VEL
LIN {X 0,Y 317.806,Z 779.953,A -85,B 0,C 180,E1 -15212.535,E2 -15212.535} C_VEL
LIN {X 0,Y 317.844,Z 779.025,A -85,B 0,C 180,E1 -15213.803,E2 -15213.803} C_VEL
LIN {X 0,Y 317.904,Z 776.697,A -85,B 0,C 180,E1 -15215.829,E2 -15215.829} C_VEL
LIN {X 0,Y 318.231,Z 772.465,A -85,B 0,C 180,E1 -15218.253,E2 -15218.253} C_VEL
LIN {X 0,Y 318.749,Z 767.862,A -85,B 0,C 180,E1 -15220.159,E2 -15220.159} C_VEL
LIN {X 0,Y 319.61,Z 760.884,A -85,B 0,C 180,E1 -15222.38,E2 -15222.38} C_VEL
LIN {X 0,Y 320.854,Z 753.332,A -85,B 0,C 180,E1 -15224.265,E2 -15224.265} C_VEL
LIN {X 0,Y 322.094,Z 744.886,A -85,B 0,C 180,E1 -15225.956,E2 -15225.956} C_VEL
LIN {X 0,Y 323.42,Z 735.043,A -85,B 0,C 180,E1 -15227.548,E2 -15227.548} C_VEL
LIN {X 0,Y 324.954,Z 724.286,A -85,B 0,C 180,E1 -15228.93,E2 -15228.93} C_VEL
LIN {X 0,Y 326.265,Z 713.743,A -85,B 0,C 180,E1 -15229.996,E2 -15229.996} C_VEL
LIN {X 0,Y 327.57,Z 701.063,A -85,B 0,C 180,E1 -15230.979,E2 -15230.979} C_VEL
LIN {X 0,Y 328.593,Z 688.21,A -85,B 0,C 180,E1 -15231.691,E2 -15231.691} C_VEL
LIN {X 0,Y 329.329,Z 675.524,A -85,B 0,C 180,E1 -15232.134,E2 -15232.134} C_VEL
LIN {X 0,Y 330.863,Z 605.526,A -85,B 0,C 180,E1 -15233.66,E2 -15233.66} C_VEL
LIN {X 0,Y 326.417,Z 571.165,A -85,B 0,C 180,E1 -15234.831,E2 -15234.831} C_VEL
LIN {X 0,Y 324.454,Z 559.346,A -85,B 0,C 180,E1 -15235.32,E2 -15235.32} C_VEL
LIN {X 0,Y 323.737,Z 549.084,A -85,B 0,C 180,E1 -15236.165,E2 -15236.165} C_VEL
LIN {X 0,Y 324.409,Z 543.296,A -85,B 0,C 180,E1 -15237.493,E2 -15237.493} C_VEL
LIN {X 0,Y 322.704,Z 534.505,A -85,B 0,C 180,E1 -15239.683,E2 -15239.683} C_VEL
LIN {X 0,Y 320.068,Z 521.989,A -85,B 0,C 180,E1 -15242.918,E2 -15242.918} C_VEL
LIN {X 0,Y 319.588,Z 519.678,A -85,B 0,C 180,E1 -15243.572,E2 -15243.572} C_VEL
LIN {X 0,Y 319.556,Z 519.662,A -85,B 0,C 180,E1 -15246.427,E2 -15246.427} C_VEL
LIN {X 0,Y 319.555,Z 519.657,A -85,B 0,C 180,E1 -15249.668,E2 -15249.668} C_VEL
LIN {X 0,Y 319.553,Z 519.672,A -85,B 0,C 180,E1 -15253.467,E2 -15253.467} C_VEL
LIN {X 0,Y 319.586,Z 519.672,A -85,B 0,C 180,E1 -15257.022,E2 -15257.022} C_VEL
LIN {X 0,Y 319.577,Z 519.676,A -85,B 0,C 180,E1 -15260.375,E2 -15260.375} C_VEL
LIN {X 0,Y 319.555,Z 519.666,A -85,B 0,C 180,E1 -15263.572,E2 -15263.572} C_VEL
LIN {X 0,Y 319.572,Z 519.678,A -85,B 0,C 180,E1 -15266.686,E2 -15266.686} C_VEL
LIN {X 0,Y 319.585,Z 519.659,A -85,B 0,C 180,E1 -15269.616,E2 -15269.616} C_VEL
LIN {X 0,Y 319.603,Z 519.672,A -85,B 0,C 180,E1 -15272.498,E2 -15272.498} C_VEL
LIN {X 0,Y 319.596,Z 519.653,A -85,B 0,C 180,E1 -15275.303,E2 -15275.303} C_VEL
LIN {X 0,Y 319.595,Z 519.675,A -85,B 0,C 180,E1 -15279.4,E2 -15279.4} C_VEL
LIN {X 0,Y 319.651,Z 519.654,A -85,B 0,C 180,E1 -15282.073,E2 -15282.073} C_VEL
LIN {X 0,Y 319.725,Z 519.654,A -85,B 0,C 180,E1 -15286.008,E2 -15286.008} C_VEL
LIN {X 0,Y 319.751,Z 519.643,A -85,B 0,C 180,E1 -15289.873,E2 -15289.873} C_VEL
LIN {X 0,Y 319.92,Z 519.61,A -85,B 0,C 180,E1 -15292.426,E2 -15292.426} C_VEL
LIN {X 0,Y 319.744,Z 519.654,A -85,B 0,C 180,E1 -15294.956,E2 -15294.956} C_VEL
LIN {X 0,Y 319.985,Z 519.619,A -85,B 0,C 180,E1 -15297.483,E2 -15297.483} C_VEL
LIN {X 0,Y 320.144,Z 519.576,A -85,B 0,C 180,E1 -15300,E2 -15300} C_VEL
LIN {X 0,Y 319.986,Z 519.618,A -85,B 0,C 180,E1 -15302.518,E2 -15302.518} C_VEL
LIN {X 0,Y 319.92,Z 519.622,A -85,B 0,C 180,E1 -15306.573,E2 -15306.573} C_VEL
LIN {X 0,Y 319.746,Z 519.645,A -85,B 0,C 180,E1 -15310.128,E2 -15310.128} C_VEL
LIN {X 0,Y 319.724,Z 519.645,A -85,B 0,C 180,E1 -15314.725,E2 -15314.725} C_VEL
LIN {X 0,Y 319.683,Z 519.662,A -85,B 0,C 180,E1 -15319.038,E2 -15319.038} C_VEL
LIN {X 0,Y 319.565,Z 519.66,A -85,B 0,C 180,E1 -15323.32,E2 -15323.32} C_VEL
LIN {X 0,Y 319.63,Z 519.669,A -85,B 0,C 180,E1 -15326.089,E2 -15326.089} C_VEL
LIN {X 0,Y 319.593,Z 519.662,A -85,B 0,C 180,E1 -15328.934,E2 -15328.934} C_VEL
LIN {X 0,Y 319.535,Z 519.682,A -85,B 0,C 180,E1 -15331.862,E2 -15331.862} C_VEL
LIN {X 0,Y 319.576,Z 519.67,A -85,B 0,C 180,E1 -15335.544,E2 -15335.544} C_VEL
LIN {X 0,Y 319.554,Z 519.681,A -85,B 0,C 180,E1 -15338.011,E2 -15338.011} C_VEL
LIN {X 0,Y 319.524,Z 519.688,A -85,B 0,C 180,E1 -15341.598,E2 -15341.598} C_VEL
LIN {X 0,Y 319.514,Z 519.686,A -85,B 0,C 180,E1 -15344.739,E2 -15344.739} C_VEL
LIN {X 0,Y 319.56,Z 519.676,A -85,B 0,C 180,E1 -15347.019,E2 -15347.019} C_VEL
LIN {X 0,Y 319.546,Z 519.68,A -85,B 0,C 180,E1 -15350.372,E2 -15350.372} C_VEL
LIN {X 0,Y 319.58,Z 519.667,A -85,B 0,C 180,E1 -15354.458,E2 -15354.458} C_VEL
LIN {X 0,Y 319.597,Z 519.695,A -85,B 0,C 180,E1 -15355.656,E2 -15355.656} C_VEL
LIN {X 0,Y 322.953,Z 532.62,A -85,B 0,C 180,E1 -15358.88,E2 -15358.88} C_VEL
LIN {X 0,Y 325.54,Z 544.38,A -85,B 0,C 180,E1 -15361.645,E2 -15361.645} C_VEL
LIN {X 0,Y 325.938,Z 547.951,A -85,B 0,C 180,E1 -15362.422,E2 -15362.422} C_VEL
LIN {X 0,Y 325.875,Z 549.981,A -85,B 0,C 180,E1 -15362.793,E2 -15362.793} C_VEL
LIN {X 0,Y 331.1,Z 576.477,A -85,B 0,C 180,E1 -15363.862,E2 -15363.862} C_VEL
LIN {X 0,Y 331.954,Z 581.398,A -85,B 0,C 180,E1 -15364.046,E2 -15364.046} C_VEL
LIN {X 0,Y 329.948,Z 661.091,A -85,B 0,C 180,E1 -15365.794,E2 -15365.794} C_VEL
LIN {X 0,Y 329.227,Z 673.749,A -85,B 0,C 180,E1 -15366.301,E2 -15366.301} C_VEL
LIN {X 0,Y 328.376,Z 686.025,A -85,B 0,C 180,E1 -15367.049,E2 -15367.049} C_VEL
LIN {X 0,Y 327.326,Z 696.931,A -85,B 0,C 180,E1 -15367.93,E2 -15367.93} C_VEL
LIN {X 0,Y 325.89,Z 708.737,A -85,B 0,C 180,E1 -15369.156,E2 -15369.156} C_VEL
LIN {X 0,Y 324.409,Z 719.184,A -85,B 0,C 180,E1 -15370.544,E2 -15370.544} C_VEL
LIN {X 0,Y 322.802,Z 729.47,A -85,B 0,C 180,E1 -15372.254,E2 -15372.254} C_VEL
LIN {X 0,Y 321.603,Z 737.193,A -85,B 0,C 180,E1 -15373.863,E2 -15373.863} C_VEL
LIN {X 0,Y 320.576,Z 744.407,A -85,B 0,C 180,E1 -15375.722,E2 -15375.722} C_VEL
LIN {X 0,Y 319.377,Z 751.221,A -85,B 0,C 180,E1 -15377.934,E2 -15377.934} C_VEL
LIN {X 0,Y 318.751,Z 755.695,A -85,B 0,C 180,E1 -15379.841,E2 -15379.841} C_VEL
LIN {X 0,Y 318.443,Z 758.04,A -85,B 0,C 180,E1 -15381.113,E2 -15381.113} C_VEL
LIN {X 0,Y 318.011,Z 761.462,A -85,B 0,C 180,E1 -15383.656,E2 -15383.656} C_VEL
LIN {X 0,Y 317.854,Z 763.181,A -85,B 0,C 180,E1 -15386.197,E2 -15386.197} C_VEL
LIN {X 0,Y 317.789,Z 763.463,A -85,B 0,C 180,E1 -15387.465,E2 -15387.465} C_VEL
LIN {X 0,Y 317.759,Z 763.358,A -85,B 0,C 180,E1 -15388.733,E2 -15388.733} C_VEL
LIN {X 0,Y 317.786,Z 762.821,A -85,B 0,C 180,E1 -15390,E2 -15390} C_VEL
LIN {X 0,Y 317.985,Z 760.591,A -85,B 0,C 180,E1 -15392.533,E2 -15392.533} C_VEL
LIN {X 0,Y 318.299,Z 757.812,A -85,B 0,C 180,E1 -15394.432,E2 -15394.432} C_VEL
LIN {X 0,Y 318.734,Z 754.018,A -85,B 0,C 180,E1 -15396.329,E2 -15396.329} C_VEL
LIN {X 0,Y 319.436,Z 748.252,A -85,B 0,C 180,E1 -15398.508,E2 -15398.508} C_VEL
LIN {X 0,Y 320.327,Z 741.706,A -85,B 0,C 180,E1 -15400.428,E2 -15400.428} C_VEL
LIN {X 0,Y 321.491,Z 733.692,A -85,B 0,C 180,E1 -15402.306,E2 -15402.306} C_VEL
LIN {X 0,Y 322.654,Z 725.478,A -85,B 0,C 180,E1 -15403.863,E2 -15403.863} C_VEL
LIN {X 0,Y 323.938,Z 715.357,A -85,B 0,C 180,E1 -15405.412,E2 -15405.412} C_VEL
LIN {X 0,Y 325.166,Z 705.385,A -85,B 0,C 180,E1 -15406.641,E2 -15406.641} C_VEL
LIN {X 0,Y 326.28,Z 694.528,A -85,B 0,C 180,E1 -15407.713,E2 -15407.713} C_VEL
LIN {X 0,Y 327.377,Z 682.4,A -85,B 0,C 180,E1 -15408.622,E2 -15408.622} C_VEL
LIN {X 0,Y 328.084,Z 669.262,A -85,B 0,C 180,E1 -15409.338,E2 -15409.338} C_VEL
LIN {X 0,Y 328.619,Z 655.853,A -85,B 0,C 180,E1 -15409.791,E2 -15409.791} C_VEL
LIN {X 0,Y 330.225,Z 579.873,A -85,B 0,C 180,E1 -15411.436,E2 -15411.436} C_VEL
LIN {X 0,Y 325.777,Z 554.921,A -85,B 0,C 180,E1 -15412.351,E2 -15412.351} C_VEL
LIN {X 0,Y 324.78,Z 549.76,A -85,B 0,C 180,E1 -15412.555,E2 -15412.555} C_VEL
LIN {X 0,Y 325.039,Z 544.569,A -85,B 0,C 180,E1 -15413.578,E2 -15413.578} C_VEL
LIN {X 0,Y 323.017,Z 533.602,A -85,B 0,C 180,E1 -15416.072,E2 -15416.072} C_VEL
LIN {X 0,Y 321.463,Z 526.909,A -85,B 0,C 180,E1 -15417.658,E2 -15417.658} C_VEL
LIN {X 0,Y 320.21,Z 524.87,A -85,B 0,C 180,E1 -15418.235,E2 -15418.235} C_VEL
LIN {X 0,Y 316.236,Z 521.991,A -85,B 0,C 180,E1 -15419.285,E2 -15419.285} C_VEL
LIN {X 0,Y 313.313,Z 520.807,A -85,B 0,C 180,E1 -15420.239,E2 -15420.239} C_VEL
LIN {X 0,Y 312.527,Z 520.556,A -85,B 0,C 180,E1 -15420.955,E2 -15420.955} C_VEL
LIN {X 0,Y 312.507,Z 520.555,A -85,B 0,C 180,E1 -15424.209,E2 -15424.209} C_VEL
LIN {X 0,Y 312.543,Z 520.553,A -85,B 0,C 180,E1 -15428.09,E2 -15428.09} C_VEL
LIN {X 0,Y 312.547,Z 520.552,A -85,B 0,C 180,E1 -15432.093,E2 -15432.093} C_VEL
LIN {X 0,Y 312.511,Z 520.546,A -85,B 0,C 180,E1 -15436.023,E2 -15436.023} C_VEL
LIN {X 0,Y 312.542,Z 520.555,A -85,B 0,C 180,E1 -15440.38,E2 -15440.38} C_VEL
LIN {X 0,Y 321.087,Z 544.655,A -85,B 0,C 180,E1 -15441.596,E2 -15441.596} C_VEL
LIN {X 0,Y 318.725,Z 621.68,A -85,B 0,C 180,E1 -15443.812,E2 -15443.812} C_VEL
LIN {X 0,Y 318.206,Z 635.006,A -85,B 0,C 180,E1 -15444.447,E2 -15444.447} C_VEL
LIN {X 0,Y 317.44,Z 648.132,A -85,B 0,C 180,E1 -15445.339,E2 -15445.339} C_VEL
LIN {X 0,Y 316.536,Z 660.676,A -85,B 0,C 180,E1 -15446.475,E2 -15446.475} C_VEL
LIN {X 0,Y 315.552,Z 672.246,A -85,B 0,C 180,E1 -15447.813,E2 -15447.813} C_VEL
LIN {X 0,Y 314.613,Z 683.497,A -85,B 0,C 180,E1 -15449.455,E2 -15449.455} C_VEL
LIN {X 0,Y 313.508,Z 693.549,A -85,B 0,C 180,E1 -15451.289,E2 -15451.289} C_VEL
LIN {X 0,Y 312.669,Z 702.284,A -85,B 0,C 180,E1 -15453.285,E2 -15453.285} C_VEL
LIN {X 0,Y 312.078,Z 709.502,A -85,B 0,C 180,E1 -15455.378,E2 -15455.378} C_VEL
LIN {X 0,Y 311.585,Z 715.523,A -85,B 0,C 180,E1 -15457.632,E2 -15457.632} C_VEL
LIN {X 0,Y 311.259,Z 719.322,A -85,B 0,C 180,E1 -15459.514,E2 -15459.514} C_VEL
LIN {X 0,Y 311.101,Z 722.354,A -85,B 0,C 180,E1 -15461.584,E2 -15461.584} C_VEL
LIN {X 0,Y 311.054,Z 723.698,A -85,B 0,C 180,E1 -15462.919,E2 -15462.919} C_VEL
LIN {X 0,Y 311.053,Z 724.584,A -85,B 0,C 180,E1 -15464.268,E2 -15464.268} C_VEL
LIN {X 0,Y 311.271,Z 725.067,A -85,B 0,C 180,E1 -15466.131,E2 -15466.131} C_VEL
LIN {X 0,Y 311.599,Z 724.54,A -85,B 0,C 180,E1 -15468.288,E2 -15468.288} C_VEL
LIN {X 0,Y 311.951,Z 723.64,A -85,B 0,C 180,E1 -15469.616,E2 -15469.616} C_VEL
LIN {X 0,Y 312.599,Z 721.457,A -85,B 0,C 180,E1 -15471.573,E2 -15471.573} C_VEL
LIN {X 0,Y 313.441,Z 718.162,A -85,B 0,C 180,E1 -15473.563,E2 -15473.563} C_VEL
LIN {X 0,Y 314.516,Z 713.77,A -85,B 0,C 180,E1 -15475.514,E2 -15475.514} C_VEL
LIN {X 0,Y 315.794,Z 708.162,A -85,B 0,C 180,E1 -15477.449,E2 -15477.449} C_VEL
LIN {X 0,Y 317.274,Z 701.079,A -85,B 0,C 180,E1 -15479.374,E2 -15479.374} C_VEL
LIN {X 0,Y 319.126,Z 692.3,A -85,B 0,C 180,E1 -15481.262,E2 -15481.262} C_VEL
LIN {X 0,Y 320.927,Z 682.229,A -85,B 0,C 180,E1 -15482.981,E2 -15482.981} C_VEL
LIN {X 0,Y 322.906,Z 670.791,A -85,B 0,C 180,E1 -15484.525,E2 -15484.525} C_VEL
LIN {X 0,Y 324.519,Z 659.279,A -85,B 0,C 180,E1 -15485.748,E2 -15485.748} C_VEL
LIN {X 0,Y 325.879,Z 647.411,A -85,B 0,C 180,E1 -15486.736,E2 -15486.736} C_VEL
LIN {X 0,Y 326.962,Z 634.461,A -85,B 0,C 180,E1 -15487.541,E2 -15487.541} C_VEL
LIN {X 0,Y 327.738,Z 621.935,A -85,B 0,C 180,E1 -15488.075,E2 -15488.075} C_VEL
LIN {X 0,Y 331.633,Z 554.281,A -85,B 0,C 180,E1 -15490.206,E2 -15490.206} C_VEL
LIN {X 0,Y 326.876,Z 544.643,A -85,B 0,C 180,E1 -15491.296,E2 -15491.296} C_VEL
LIN {X 0,Y 320.499,Z 534.12,A -85,B 0,C 180,E1 -15492.804,E2 -15492.804} C_VEL
LIN {X 0,Y 315.687,Z 526.873,A -85,B 0,C 180,E1 -15494.034,E2 -15494.034} C_VEL
LIN {X 0,Y 313.495,Z 523.398,A -85,B 0,C 180,E1 -15494.673,E2 -15494.673} C_VEL
LIN {X 0,Y 312.63,Z 520.542,A -85,B 0,C 180,E1 -15496.656,E2 -15496.656} C_VEL
LIN {X 0,Y 312.582,Z 520.547,A -85,B 0,C 180,E1 -15499.71,E2 -15499.71} C_VEL
LIN {X 0,Y 312.539,Z 520.556,A -85,B 0,C 180,E1 -15502.789,E2 -15502.789} C_VEL
LIN {X 0,Y 312.577,Z 520.548,A -85,B 0,C 180,E1 -15506.723,E2 -15506.723} C_VEL
LIN {X 0,Y 312.54,Z 520.546,A -85,B 0,C 180,E1 -15509.65,E2 -15509.65} C_VEL
LIN {X 0,Y 312.514,Z 520.55,A -85,B 0,C 180,E1 -15513.689,E2 -15513.689} C_VEL
LIN {X 0,Y 312.515,Z 520.556,A -85,B 0,C 180,E1 -15517.386,E2 -15517.386} C_VEL
LIN {X 0,Y 312.486,Z 520.559,A -85,B 0,C 180,E1 -15520.71,E2 -15520.71} C_VEL
LIN {X 0,Y 312.469,Z 520.562,A -85,B 0,C 180,E1 -15524.206,E2 -15524.206} C_VEL
LIN {X 0,Y 312.523,Z 520.696,A -85,B 0,C 180,E1 -15527.357,E2 -15527.357} C_VEL
LIN {X 0,Y 314.265,Z 526.262,A -85,B 0,C 180,E1 -15530.457,E2 -15530.457} C_VEL
LIN {X 0,Y 316.055,Z 532.018,A -85,B 0,C 180,E1 -15533.18,E2 -15533.18} C_VEL
LIN {X 0,Y 317.714,Z 538.352,A -85,B 0,C 180,E1 -15535.77,E2 -15535.77} C_VEL
LIN {X 0,Y 319.561,Z 546.511,A -85,B 0,C 180,E1 -15538.727,E2 -15538.727} C_VEL
LIN {X 0,Y 320.589,Z 552.474,A -85,B 0,C 180,E1 -15540.651,E2 -15540.651} C_VEL
LIN {X 0,Y 322.226,Z 558.166,A -85,B 0,C 180,E1 -15541.166,E2 -15541.166} C_VEL
LIN {X 0,Y 325.414,Z 573.486,A -85,B 0,C 180,E1 -15542.311,E2 -15542.311} C_VEL
LIN {X 0,Y 327.745,Z 588.726,A -85,B 0,C 180,E1 -15543.258,E2 -15543.258} C_VEL
LIN {X 0,Y 329.185,Z 604.817,A -85,B 0,C 180,E1 -15544.091,E2 -15544.091} C_VEL
LIN {X 0,Y 329.156,Z 610.594,A -85,B 0,C 180,E1 -15544.307,E2 -15544.307} C_VEL
LIN {X 0,Y 326.054,Z 666.16,A -85,B 0,C 180,E1 -15546.036,E2 -15546.036} C_VEL
LIN {X 0,Y 324.646,Z 680.59,A -85,B 0,C 180,E1 -15546.73,E2 -15546.73} C_VEL
LIN {X 0,Y 322.906,Z 693.559,A -85,B 0,C 180,E1 -15547.612,E2 -15547.612} C_VEL
LIN {X 0,Y 320.799,Z 706.9,A -85,B 0,C 180,E1 -15548.81,E2 -15548.81} C_VEL
LIN {X 0,Y 318.809,Z 718.696,A -85,B 0,C 180,E1 -15550.189,E2 -15550.189} C_VEL
LIN {X 0,Y 316.984,Z 728.375,A -85,B 0,C 180,E1 -15551.583,E2 -15551.583} C_VEL
LIN {X 0,Y 314.173,Z 746.686,A -85,B 0,C 180,E1 -15554.761,E2 -15554.761} C_VEL
LIN {X 0,Y 312.932,Z 755.594,A -85,B 0,C 180,E1 -15556.691,E2 -15556.691} C_VEL
LIN {X 0,Y 311.975,Z 762.734,A -85,B 0,C 180,E1 -15558.632,E2 -15558.632} C_VEL
LIN {X 0,Y 311.28,Z 769.209,A -85,B 0,C 180,E1 -15560.907,E2 -15560.907} C_VEL
LIN {X 0,Y 310.933,Z 773.465,A -85,B 0,C 180,E1 -15562.859,E2 -15562.859} C_VEL
LIN {X 0,Y 310.772,Z 776.638,A -85,B 0,C 180,E1 -15564.81,E2 -15564.81} C_VEL
LIN {X 0,Y 310.754,Z 778.211,A -85,B 0,C 180,E1 -15566.11,E2 -15566.11} C_VEL
LIN {X 0,Y 310.727,Z 779.347,A -85,B 0,C 180,E1 -15567.407,E2 -15567.407} C_VEL
LIN {X 0,Y 310.689,Z 780.049,A -85,B 0,C 180,E1 -15568.704,E2 -15568.704} C_VEL
LIN {X 0,Y 310.699,Z 780.362,A -85,B 0,C 180,E1 -15570,E2 -15570} C_VEL
LIN {X 0,Y 310.679,Z 780.284,A -85,B 0,C 180,E1 -15571.296,E2 -15571.296} C_VEL
LIN {X 0,Y 310.727,Z 779.774,A -85,B 0,C 180,E1 -15572.593,E2 -15572.593} C_VEL
LIN {X 0,Y 310.754,Z 778.85,A -85,B 0,C 180,E1 -15573.89,E2 -15573.89} C_VEL
LIN {X 0,Y 310.827,Z 776.748,A -85,B 0,C 180,E1 -15575.806,E2 -15575.806} C_VEL
LIN {X 0,Y 311.046,Z 773.567,A -85,B 0,C 180,E1 -15577.791,E2 -15577.791} C_VEL
LIN {X 0,Y 311.504,Z 769.362,A -85,B 0,C 180,E1 -15579.742,E2 -15579.742} C_VEL
LIN {X 0,Y 312.335,Z 762.953,A -85,B 0,C 180,E1 -15582.013,E2 -15582.013} C_VEL
LIN {X 0,Y 313.489,Z 755.924,A -85,B 0,C 180,E1 -15583.945,E2 -15583.945} C_VEL
LIN {X 0,Y 314.804,Z 747.515,A -85,B 0,C 180,E1 -15585.794,E2 -15585.794} C_VEL
LIN {X 0,Y 316.222,Z 738.118,A -85,B 0,C 180,E1 -15587.459,E2 -15587.459} C_VEL
LIN {X 0,Y 317.666,Z 728.113,A -85,B 0,C 180,E1 -15588.878,E2 -15588.878} C_VEL
LIN {X 0,Y 319.204,Z 716.991,A -85,B 0,C 180,E1 -15590.121,E2 -15590.121} C_VEL
LIN {X 0,Y 320.61,Z 704.484,A -85,B 0,C 180,E1 -15591.204,E2 -15591.204} C_VEL
LIN {X 0,Y 321.803,Z 691.51,A -85,B 0,C 180,E1 -15592.004,E2 -15592.004} C_VEL
LIN {X 0,Y 322.631,Z 678.724,A -85,B 0,C 180,E1 -15592.535,E2 -15592.535} C_VEL
LIN {X 0,Y 324.065,Z 622.329,A -85,B 0,C 180,E1 -15593.807,E2 -15593.807} C_VEL
LIN {X 0,Y 324.239,Z 604.927,A -85,B 0,C 180,E1 -15594.207,E2 -15594.207} C_VEL
LIN {X 0,Y 319.766,Z 570.521,A -85,B 0,C 180,E1 -15595.42,E2 -15595.42} C_VEL
LIN {X 0,Y 317.933,Z 559.601,A -85,B 0,C 180,E1 -15595.876,E2 -15595.876} C_VEL
LIN {X 0,Y 317.061,Z 547.185,A -85,B 0,C 180,E1 -15596.937,E2 -15596.937} C_VEL
LIN {X 0,Y 317.358,Z 543.899,A -85,B 0,C 180,E1 -15597.713,E2 -15597.713} C_VEL
LIN {X 0,Y 314.853,Z 531.547,A -85,B 0,C 180,E1 -15600.889,E2 -15600.889} C_VEL
LIN {X 0,Y 312.554,Z 520.553,A -85,B 0,C 180,E1 -15603.853,E2 -15603.853} C_VEL
LIN {X 0,Y 312.517,Z 520.523,A -85,B 0,C 180,E1 -15607.385,E2 -15607.385} C_VEL
LIN {X 0,Y 312.487,Z 520.556,A -85,B 0,C 180,E1 -15610.708,E2 -15610.708} C_VEL
LIN {X 0,Y 312.472,Z 520.555,A -85,B 0,C 180,E1 -15614.205,E2 -15614.205} C_VEL
LIN {X 0,Y 312.528,Z 520.544,A -85,B 0,C 180,E1 -15617.908,E2 -15617.908} C_VEL
LIN {X 0,Y 312.552,Z 520.548,A -85,B 0,C 180,E1 -15621.905,E2 -15621.905} C_VEL
LIN {X 0,Y 312.501,Z 520.558,A -85,B 0,C 180,E1 -15625.789,E2 -15625.789} C_VEL
LIN {X 0,Y 312.518,Z 520.54,A -85,B 0,C 180,E1 -15628.853,E2 -15628.853} C_VEL
LIN {X 0,Y 312.569,Z 520.548,A -85,B 0,C 180,E1 -15631.824,E2 -15631.824} C_VEL
LIN {X 0,Y 312.578,Z 520.534,A -85,B 0,C 180,E1 -15634.71,E2 -15634.71} C_VEL
LIN {X 0,Y 312.53,Z 520.552,A -85,B 0,C 180,E1 -15638.912,E2 -15638.912} C_VEL
LIN {X 0,Y 312.631,Z 520.53,A -85,B 0,C 180,E1 -15641.656,E2 -15641.656} C_VEL
LIN {X 0,Y 312.687,Z 520.528,A -85,B 0,C 180,E1 -15645.686,E2 -15645.686} C_VEL
LIN {X 0,Y 312.696,Z 520.522,A -85,B 0,C 180,E1 -15649.642,E2 -15649.642} C_VEL
LIN {X 0,Y 312.861,Z 520.488,A -85,B 0,C 180,E1 -15652.254,E2 -15652.254} C_VEL
LIN {X 0,Y 312.714,Z 520.529,A -85,B 0,C 180,E1 -15654.843,E2 -15654.843} C_VEL
LIN {X 0,Y 312.985,Z 520.478,A -85,B 0,C 180,E1 -15658.714,E2 -15658.714} C_VEL
LIN {X 0,Y 312.985,Z 520.475,A -85,B 0,C 180,E1 -15661.287,E2 -15661.287} C_VEL
LIN {X 0,Y 312.714,Z 520.53,A -85,B 0,C 180,E1 -15665.158,E2 -15665.158} C_VEL
LIN {X 0,Y 312.847,Z 520.49,A -85,B 0,C 180,E1 -15667.747,E2 -15667.747} C_VEL
LIN {X 0,Y 312.662,Z 520.538,A -85,B 0,C 180,E1 -15671.672,E2 -15671.672} C_VEL
LIN {X 0,Y 312.694,Z 520.518,A -85,B 0,C 180,E1 -15674.888,E2 -15674.888} C_VEL
LIN {X 0,Y 312.624,Z 520.544,A -85,B 0,C 180,E1 -15679.237,E2 -15679.237} C_VEL
LIN {X 0,Y 312.54,Z 520.536,A -85,B 0,C 180,E1 -15682.79,E2 -15682.79} C_VEL
LIN {X 0,Y 312.578,Z 520.55,A -85,B 0,C 180,E1 -15686.724,E2 -15686.724} C_VEL
LIN {X 0,Y 312.546,Z 520.537,A -85,B 0,C 180,E1 -15689.65,E2 -15689.65} C_VEL
LIN {X 0,Y 312.516,Z 520.551,A -85,B 0,C 180,E1 -15693.69,E2 -15693.69} C_VEL
LIN {X 0,Y 312.523,Z 520.56,A -85,B 0,C 180,E1 -15697.386,E2 -15697.386} C_VEL
LIN {X 0,Y 312.488,Z 520.559,A -85,B 0,C 180,E1 -15700.71,E2 -15700.71} C_VEL
LIN {X 0,Y 312.471,Z 520.56,A -85,B 0,C 180,E1 -15704.207,E2 -15704.207} C_VEL
LIN {X 0,Y 312.485,Z 520.561,A -85,B 0,C 180,E1 -15707.919,E2 -15707.919} C_VEL
LIN {X 0,Y 312.498,Z 520.562,A -85,B 0,C 180,E1 -15710.972,E2 -15710.972} C_VEL
LIN {X 0,Y 312.531,Z 520.543,A -85,B 0,C 180,E1 -15715.011,E2 -15715.011} C_VEL
LIN {X 0,Y 315.819,Z 532.896,A -85,B 0,C 180,E1 -15718.205,E2 -15718.205} C_VEL
LIN {X 0,Y 318.683,Z 545.533,A -85,B 0,C 180,E1 -15721.238,E2 -15721.238} C_VEL
LIN {X 0,Y 319.218,Z 549.928,A -85,B 0,C 180,E1 -15722.197,E2 -15722.197} C_VEL
LIN {X 0,Y 324.716,Z 577.652,A -85,B 0,C 180,E1 -15723.361,E2 -15723.361} C_VEL
LIN {X 0,Y 325.495,Z 582.991,A -85,B 0,C 180,E1 -15723.555,E2 -15723.555} C_VEL
LIN {X 0,Y 323.486,Z 660.386,A -85,B 0,C 180,E1 -15725.278,E2 -15725.278} C_VEL
LIN {X 0,Y 322.723,Z 673.726,A -85,B 0,C 180,E1 -15725.809,E2 -15725.809} C_VEL
LIN {X 0,Y 321.825,Z 685.856,A -85,B 0,C 180,E1 -15726.555,E2 -15726.555} C_VEL
LIN {X 0,Y 320.561,Z 698.538,A -85,B 0,C 180,E1 -15727.609,E2 -15727.609} C_VEL
LIN {X 0,Y 319.068,Z 709.973,A -85,B 0,C 180,E1 -15728.858,E2 -15728.858} C_VEL
LIN {X 0,Y 317.532,Z 720.245,A -85,B 0,C 180,E1 -15730.274,E2 -15730.274} C_VEL
LIN {X 0,Y 316.016,Z 729.524,A -85,B 0,C 180,E1 -15731.86,E2 -15731.86} C_VEL
LIN {X 0,Y 314.704,Z 737.513,A -85,B 0,C 180,E1 -15733.558,E2 -15733.558} C_VEL
LIN {X 0,Y 313.667,Z 744.51,A -85,B 0,C 180,E1 -15735.401,E2 -15735.401} C_VEL
LIN {X 0,Y 312.419,Z 751.342,A -85,B 0,C 180,E1 -15737.661,E2 -15737.661} C_VEL
LIN {X 0,Y 311.733,Z 755.834,A -85,B 0,C 180,E1 -15739.61,E2 -15739.61} C_VEL
LIN {X 0,Y 311.399,Z 758.191,A -85,B 0,C 180,E1 -15740.91,E2 -15740.91} C_VEL
LIN {X 0,Y 310.927,Z 761.626,A -85,B 0,C 180,E1 -15743.511,E2 -15743.511} C_VEL
LIN {X 0,Y 310.796,Z 762.697,A -85,B 0,C 180,E1 -15744.811,E2 -15744.811} C_VEL
LIN {X 0,Y 310.765,Z 763.363,A -85,B 0,C 180,E1 -15746.11,E2 -15746.11} C_VEL
LIN {X 0,Y 310.712,Z 763.65,A -85,B 0,C 180,E1 -15747.407,E2 -15747.407} C_VEL
LIN {X 0,Y 310.673,Z 763.555,A -85,B 0,C 180,E1 -15748.704,E2 -15748.704} C_VEL
LIN {X 0,Y 310.696,Z 763.027,A -85,B 0,C 180,E1 -15750,E2 -15750} C_VEL
LIN {X 0,Y 310.905,Z 760.81,A -85,B 0,C 180,E1 -15752.591,E2 -15752.591} C_VEL
LIN {X 0,Y 311.242,Z 758.042,A -85,B 0,C 180,E1 -15754.533,E2 -15754.533} C_VEL
LIN {X 0,Y 311.691,Z 754.262,A -85,B 0,C 180,E1 -15756.473,E2 -15756.473} C_VEL
LIN {X 0,Y 312.303,Z 749.365,A -85,B 0,C 180,E1 -15758.411,E2 -15758.411} C_VEL
LIN {X 0,Y 313.166,Z 743.187,A -85,B 0,C 180,E1 -15760.342,E2 -15760.342} C_VEL
LIN {X 0,Y 314.336,Z 735.438,A -85,B 0,C 180,E1 -15762.263,E2 -15762.263} C_VEL
LIN {X 0,Y 315.763,Z 725.803,A -85,B 0,C 180,E1 -15764.171,E2 -15764.171} C_VEL
LIN {X 0,Y 317.115,Z 715.714,A -85,B 0,C 180,E1 -15765.752,E2 -15765.752} C_VEL
LIN {X 0,Y 318.381,Z 705.775,A -85,B 0,C 180,E1 -15767.006,E2 -15767.006} C_VEL
LIN {X 0,Y 319.555,Z 694.962,A -85,B 0,C 180,E1 -15768.098,E2 -15768.098} C_VEL
LIN {X 0,Y 320.675,Z 682.939,A -85,B 0,C 180,E1 -15769.026,E2 -15769.026} C_VEL
LIN {X 0,Y 321.41,Z 669.925,A -85,B 0,C 180,E1 -15769.756,E2 -15769.756} C_VEL
LIN {X 0,Y 321.972,Z 656.608,A -85,B 0,C 180,E1 -15770.226,E2 -15770.226} C_VEL
LIN {X 0,Y 323.647,Z 580.556,A -85,B 0,C 180,E1 -15771.906,E2 -15771.906} C_VEL
LIN {X 0,Y 318.446,Z 551.702,A -85,B 0,C 180,E1 -15773.004,E2 -15773.004} C_VEL
LIN {X 0,Y 318.102,Z 549.85,A -85,B 0,C 180,E1 -15773.095,E2 -15773.095} C_VEL
LIN {X 0,Y 318.113,Z 545.031,A -85,B 0,C 180,E1 -15774.075,E2 -15774.075} C_VEL
LIN {X 0,Y 315.573,Z 532.38,A -85,B 0,C 180,E1 -15777.022,E2 -15777.022} C_VEL
LIN {X 0,Y 312.589,Z 520.553,A -85,B 0,C 180,E1 -15779.969,E2 -15779.969} C_VEL
LIN {X 0,Y 312.527,Z 520.556,A -85,B 0,C 180,E1 -15780.955,E2 -15780.955} C_VEL
LIN {X 0,Y 311.853,Z 520.643,A -85,B 0,C 180,E1 -15782.03,E2 -15782.03} C_VEL
LIN {X 0,Y 309.005,Z 520.99,A -85,B 0,C 180,E1 -15783.781,E2 -15783.781} C_VEL
LIN {X 0,Y 306.6,Z 521.295,A -85,B 0,C 180,E1 -15785.201,E2 -15785.201} C_VEL
LIN {X 0,Y 305.576,Z 521.416,A -85,B 0,C 180,E1 -15786.3,E2 -15786.3} C_VEL
LIN {X 0,Y 305.497,Z 521.424,A -85,B 0,C 180,E1 -15786.672,E2 -15786.672} C_VEL
LIN {X 0,Y 305.484,Z 521.422,A -85,B 0,C 180,E1 -15790.605,E2 -15790.605} C_VEL
LIN {X 0,Y 305.489,Z 521.429,A -85,B 0,C 180,E1 -15793.642,E2 -15793.642} C_VEL
LIN {X 0,Y 305.461,Z 521.436,A -85,B 0,C 180,E1 -15797.412,E2 -15797.412} C_VEL
LIN {X 0,Y 305.479,Z 521.433,A -85,B 0,C 180,E1 -15800.005,E2 -15800.005} C_VEL
LIN {X 0,Y 314.169,Z 545.904,A -85,B 0,C 180,E1 -15801.28,E2 -15801.28} C_VEL
LIN {X 0,Y 311.804,Z 622.451,A -85,B 0,C 180,E1 -15803.548,E2 -15803.548} C_VEL
LIN {X 0,Y 311.284,Z 635.579,A -85,B 0,C 180,E1 -15804.192,E2 -15804.192} C_VEL
LIN {X 0,Y 310.589,Z 647.435,A -85,B 0,C 180,E1 -15805.001,E2 -15805.001} C_VEL
LIN {X 0,Y 309.582,Z 660.672,A -85,B 0,C 180,E1 -15806.207,E2 -15806.207} C_VEL
LIN {X 0,Y 308.647,Z 671.822,A -85,B 0,C 180,E1 -15807.501,E2 -15807.501} C_VEL
LIN {X 0,Y 307.71,Z 682.613,A -85,B 0,C 180,E1 -15809.076,E2 -15809.076} C_VEL
LIN {X 0,Y 306.61,Z 692.53,A -85,B 0,C 180,E1 -15810.855,E2 -15810.855} C_VEL
LIN {X 0,Y 305.841,Z 700.547,A -85,B 0,C 180,E1 -15812.639,E2 -15812.639} C_VEL
LIN {X 0,Y 305.13,Z 708.268,A -85,B 0,C 180,E1 -15814.779,E2 -15814.779} C_VEL
LIN {X 0,Y 304.63,Z 714.313,A -85,B 0,C 180,E1 -15816.908,E2 -15816.908} C_VEL
LIN {X 0,Y 304.251,Z 718.877,A -85,B 0,C 180,E1 -15819.02,E2 -15819.02} C_VEL
LIN {X 0,Y 304.026,Z 722.535,A -85,B 0,C 180,E1 -15821.397,E2 -15821.397} C_VEL
LIN {X 0,Y 303.976,Z 724.885,A -85,B 0,C 180,E1 -15823.892,E2 -15823.892} C_VEL
LIN {X 0,Y 304.179,Z 725.671,A -85,B 0,C 180,E1 -15826.019,E2 -15826.019} C_VEL
LIN {X 0,Y 304.475,Z 725.422,A -85,B 0,C 180,E1 -15828.01,E2 -15828.01} C_VEL
LIN {X 0,Y 304.827,Z 724.677,A -85,B 0,C 180,E1 -15829.371,E2 -15829.371} C_VEL
LIN {X 0,Y 305.533,Z 722.591,A -85,B 0,C 180,E1 -15831.524,E2 -15831.524} C_VEL
LIN {X 0,Y 306.33,Z 719.804,A -85,B 0,C 180,E1 -15833.413,E2 -15833.413} C_VEL
LIN {X 0,Y 307.45,Z 715.745,A -85,B 0,C 180,E1 -15835.411,E2 -15835.411} C_VEL
LIN {X 0,Y 308.776,Z 710.488,A -85,B 0,C 180,E1 -15837.391,E2 -15837.391} C_VEL
LIN {X 0,Y 310.317,Z 703.873,A -85,B 0,C 180,E1 -15839.351,E2 -15839.351} C_VEL
LIN {X 0,Y 312.154,Z 695.609,A -85,B 0,C 180,E1 -15841.29,E2 -15841.29} C_VEL
LIN {X 0,Y 313.876,Z 687.185,A -85,B 0,C 180,E1 -15842.887,E2 -15842.887} C_VEL
LIN {X 0,Y 315.604,Z 677.995,A -85,B 0,C 180,E1 -15844.31,E2 -15844.31} C_VEL
LIN {X 0,Y 317.494,Z 666.694,A -85,B 0,C 180,E1 -15845.717,E2 -15845.717} C_VEL
LIN {X 0,Y 319.169,Z 654.904,A -85,B 0,C 180,E1 -15846.855,E2 -15846.855} C_VEL
LIN {X 0,Y 320.492,Z 642.456,A -85,B 0,C 180,E1 -15847.798,E2 -15847.798} C_VEL
LIN {X 0,Y 321.468,Z 629.267,A -85,B 0,C 180,E1 -15848.525,E2 -15848.525} C_VEL
LIN {X 0,Y 322.95,Z 603.329,A -85,B 0,C 180,E1 -15849.416,E2 -15849.416} C_VEL
LIN {X 0,Y 325.961,Z 556.705,A -85,B 0,C 180,E1 -15850.916,E2 -15850.916} C_VEL
LIN {X 0,Y 322.003,Z 548.739,A -85,B 0,C 180,E1 -15851.89,E2 -15851.89} C_VEL
LIN {X 0,Y 316.557,Z 539.465,A -85,B 0,C 180,E1 -15853.249,E2 -15853.249} C_VEL
LIN {X 0,Y 311.756,Z 532.163,A -85,B 0,C 180,E1 -15854.528,E2 -15854.528} C_VEL
LIN {X 0,Y 309.137,Z 528.417,A -85,B 0,C 180,E1 -15855.274,E2 -15855.274} C_VEL
LIN {X 0,Y 306.809,Z 525.277,A -85,B 0,C 180,E1 -15855.955,E2 -15855.955} C_VEL
LIN {X 0,Y 306.475,Z 524.514,A -85,B 0,C 180,E1 -15856.143,E2 -15856.143} C_VEL
LIN {X 0,Y 305.599,Z 521.418,A -85,B 0,C 180,E1 -15858.608,E2 -15858.608} C_VEL
LIN {X 0,Y 305.484,Z 521.432,A -85,B 0,C 180,E1 -15863.041,E2 -15863.041} C_VEL
LIN {X 0,Y 305.548,Z 521.421,A -85,B 0,C 180,E1 -15866.23,E2 -15866.23} C_VEL
LIN {X 0,Y 305.49,Z 521.427,A -85,B 0,C 180,E1 -15869.05,E2 -15869.05} C_VEL
LIN {X 0,Y 305.46,Z 521.43,A -85,B 0,C 180,E1 -15873.517,E2 -15873.517} C_VEL
LIN {X 0,Y 305.467,Z 521.432,A -85,B 0,C 180,E1 -15876.74,E2 -15876.74} C_VEL
LIN {X 0,Y 305.45,Z 521.435,A -85,B 0,C 180,E1 -15880.6,E2 -15880.6} C_VEL
LIN {X 0,Y 305.415,Z 521.442,A -85,B 0,C 180,E1 -15884.493,E2 -15884.493} C_VEL
LIN {X 0,Y 305.457,Z 521.656,A -85,B 0,C 180,E1 -15885.5,E2 -15885.5} C_VEL
LIN {X 0,Y 306.908,Z 526.055,A -85,B 0,C 180,E1 -15888.389,E2 -15888.389} C_VEL
LIN {X 0,Y 309.183,Z 533.119,A -85,B 0,C 180,E1 -15892.141,E2 -15892.141} C_VEL
LIN {X 0,Y 311.285,Z 541.233,A -85,B 0,C 180,E1 -15895.638,E2 -15895.638} C_VEL
LIN {X 0,Y 313.004,Z 549.083,A -85,B 0,C 180,E1 -15898.564,E2 -15898.564} C_VEL
LIN {X 0,Y 313.499,Z 551.586,A -85,B 0,C 180,E1 -15899.371,E2 -15899.371} C_VEL
LIN {X 0,Y 315.84,Z 556.639,A -85,B 0,C 180,E1 -15900.039,E2 -15900.039} C_VEL
LIN {X 0,Y 317.087,Z 561.003,A -85,B 0,C 180,E1 -15900.454,E2 -15900.454} C_VEL
LIN {X 0,Y 320.066,Z 575.95,A -85,B 0,C 180,E1 -15901.607,E2 -15901.607} C_VEL
LIN {X 0,Y 322.443,Z 592.697,A -85,B 0,C 180,E1 -15902.684,E2 -15902.684} C_VEL
LIN {X 0,Y 323.623,Z 608.527,A -85,B 0,C 180,E1 -15903.494,E2 -15903.494} C_VEL
LIN {X 0,Y 320.092,Z 665.958,A -85,B 0,C 180,E1 -15905.345,E2 -15905.345} C_VEL
LIN {X 0,Y 318.696,Z 679.58,A -85,B 0,C 180,E1 -15906.01,E2 -15906.01} C_VEL
LIN {X 0,Y 316.734,Z 693.57,A -85,B 0,C 180,E1 -15906.979,E2 -15906.979} C_VEL
LIN {X 0,Y 314.803,Z 705.239,A -85,B 0,C 180,E1 -15908.041,E2 -15908.041} C_VEL
LIN {X 0,Y 312.617,Z 717.132,A -85,B 0,C 180,E1 -15909.436,E2 -15909.436} C_VEL
LIN {X 0,Y 310.664,Z 726.899,A -85,B 0,C 180,E1 -15910.851,E2 -15910.851} C_VEL
LIN {X 0,Y 308.927,Z 735.968,A -85,B 0,C 180,E1 -15912.457,E2 -15912.457} C_VEL
LIN {X 0,Y 306.829,Z 749.622,A -85,B 0,C 180,E1 -15915.068,E2 -15915.068} C_VEL
LIN {X 0,Y 305.622,Z 757.874,A -85,B 0,C 180,E1 -15917.044,E2 -15917.044} C_VEL
LIN {X 0,Y 304.858,Z 763.497,A -85,B 0,C 180,E1 -15918.7,E2 -15918.7} C_VEL
LIN {X 0,Y 304.234,Z 768.97,A -85,B 0,C 180,E1 -15920.694,E2 -15920.694} C_VEL
LIN {X 0,Y 303.853,Z 773.237,A -85,B 0,C 180,E1 -15922.692,E2 -15922.692} C_VEL
LIN {X 0,Y 303.685,Z 776.42,A -85,B 0,C 180,E1 -15924.689,E2 -15924.689} C_VEL
LIN {X 0,Y 303.667,Z 777.999,A -85,B 0,C 180,E1 -15926.019,E2 -15926.019} C_VEL
LIN {X 0,Y 303.65,Z 779.144,A -85,B 0,C 180,E1 -15927.347,E2 -15927.347} C_VEL
LIN {X 0,Y 303.605,Z 779.851,A -85,B 0,C 180,E1 -15928.674,E2 -15928.674} C_VEL
LIN {X 0,Y 303.612,Z 780.169,A -85,B 0,C 180,E1 -15930,E2 -15930} C_VEL
LIN {X 0,Y 303.595,Z 780.096,A -85,B 0,C 180,E1 -15931.326,E2 -15931.326} C_VEL
LIN {X 0,Y 303.65,Z 779.595,A -85,B 0,C 180,E1 -15932.653,E2 -15932.653} C_VEL
LIN {X 0,Y 303.668,Z 778.676,A -85,B 0,C 180,E1 -15933.981,E2 -15933.981} C_VEL
LIN {X 0,Y 303.729,Z 776.85,A -85,B 0,C 180,E1 -15935.744,E2 -15935.744} C_VEL
LIN {X 0,Y 304.003,Z 773.414,A -85,B 0,C 180,E1 -15937.973,E2 -15937.973} C_VEL
LIN {X 0,Y 304.467,Z 769.22,A -85,B 0,C 180,E1 -15939.969,E2 -15939.969} C_VEL
LIN {X 0,Y 305.371,Z 762.824,A -85,B 0,C 180,E1 -15942.291,E2 -15942.291} C_VEL
LIN {X 0,Y 306.586,Z 755.817,A -85,B 0,C 180,E1 -15944.266,E2 -15944.266} C_VEL
LIN {X 0,Y 307.944,Z 747.588,A -85,B 0,C 180,E1 -15946.121,E2 -15946.121} C_VEL
LIN {X 0,Y 309.439,Z 738.051,A -85,B 0,C 180,E1 -15947.855,E2 -15947.855} C_VEL
LIN {X 0,Y 310.968,Z 728.089,A -85,B 0,C 180,E1 -15949.301,E2 -15949.301} C_VEL
LIN {X 0,Y 312.553,Z 717.005,A -85,B 0,C 180,E1 -15950.569,E2 -15950.569} C_VEL
LIN {X 0,Y 313.998,Z 704.567,A -85,B 0,C 180,E1 -15951.672,E2 -15951.672} C_VEL
LIN {X 0,Y 315.25,Z 691.72,A -85,B 0,C 180,E1 -15952.486,E2 -15952.486} C_VEL
LIN {X 0,Y 316.107,Z 679.134,A -85,B 0,C 180,E1 -15953.026,E2 -15953.026} C_VEL
LIN {X 0,Y 316.885,Z 652.762,A -85,B 0,C 180,E1 -15953.66,E2 -15953.66} C_VEL
LIN {X 0,Y 317.887,Z 606.325,A -85,B 0,C 180,E1 -15954.708,E2 -15954.708} C_VEL
LIN {X 0,Y 313.568,Z 572.463,A -85,B 0,C 180,E1 -15955.93,E2 -15955.93} C_VEL
LIN {X 0,Y 311.411,Z 559.389,A -85,B 0,C 180,E1 -15956.488,E2 -15956.488} C_VEL
LIN {X 0,Y 310.393,Z 545.142,A -85,B 0,C 180,E1 -15957.776,E2 -15957.776} C_VEL
LIN {X 0,Y 307.646,Z 531.693,A -85,B 0,C 180,E1 -15961.312,E2 -15961.312} C_VEL
LIN {X 0,Y 305.507,Z 521.43,A -85,B 0,C 180,E1 -15964.179,E2 -15964.179} C_VEL
LIN {X 0,Y 305.47,Z 521.409,A -85,B 0,C 180,E1 -15966.739,E2 -15966.739} C_VEL
LIN {X 0,Y 305.452,Z 521.431,A -85,B 0,C 180,E1 -15970.599,E2 -15970.599} C_VEL
LIN {X 0,Y 305.423,Z 521.434,A -85,B 0,C 180,E1 -15974.493,E2 -15974.493} C_VEL
LIN {X 0,Y 305.475,Z 521.421,A -85,B 0,C 180,E1 -15978.149,E2 -15978.149} C_VEL
LIN {X 0,Y 305.514,Z 521.426,A -85,B 0,C 180,E1 -15981.603,E2 -15981.603} C_VEL
LIN {X 0,Y 305.458,Z 521.429,A -85,B 0,C 180,E1 -15984.886,E2 -15984.886} C_VEL
LIN {X 0,Y 305.446,Z 521.424,A -85,B 0,C 180,E1 -15988.355,E2 -15988.355} C_VEL
LIN {X 0,Y 305.515,Z 521.421,A -85,B 0,C 180,E1 -15991.113,E2 -15991.113} C_VEL
LIN {X 0,Y 305.565,Z 521.415,A -85,B 0,C 180,E1 -15994.088,E2 -15994.088} C_VEL
LIN {X 0,Y 305.475,Z 521.428,A -85,B 0,C 180,E1 -15998.401,E2 -15998.401} C_VEL
LIN {X 0,Y 305.582,Z 521.411,A -85,B 0,C 180,E1 -16001.217,E2 -16001.217} C_VEL
LIN {X 0,Y 305.642,Z 521.4,A -85,B 0,C 180,E1 -16005.349,E2 -16005.349} C_VEL
LIN {X 0,Y 305.633,Z 521.404,A -85,B 0,C 180,E1 -16009.4,E2 -16009.4} C_VEL
LIN {X 0,Y 305.802,Z 521.365,A -85,B 0,C 180,E1 -16012.074,E2 -16012.074} C_VEL
LIN {X 0,Y 305.684,Z 521.403,A -85,B 0,C 180,E1 -16014.724,E2 -16014.724} C_VEL
LIN {X 0,Y 305.952,Z 521.354,A -85,B 0,C 180,E1 -16018.684,E2 -16018.684} C_VEL
LIN {X 0,Y 305.952,Z 521.351,A -85,B 0,C 180,E1 -16021.317,E2 -16021.317} C_VEL
LIN {X 0,Y 305.685,Z 521.404,A -85,B 0,C 180,E1 -16025.277,E2 -16025.277} C_VEL
LIN {X 0,Y 305.791,Z 521.367,A -85,B 0,C 180,E1 -16027.927,E2 -16027.927} C_VEL
LIN {X 0,Y 305.597,Z 521.417,A -85,B 0,C 180,E1 -16031.946,E2 -16031.946} C_VEL
LIN {X 0,Y 305.631,Z 521.395,A -85,B 0,C 180,E1 -16035.035,E2 -16035.035} C_VEL
LIN {X 0,Y 305.571,Z 521.423,A -85,B 0,C 180,E1 -16039.445,E2 -16039.445} C_VEL
LIN {X 0,Y 305.485,Z 521.413,A -85,B 0,C 180,E1 -16043.042,E2 -16043.042} C_VEL
LIN {X 0,Y 305.549,Z 521.423,A -85,B 0,C 180,E1 -16046.23,E2 -16046.23} C_VEL
LIN {X 0,Y 305.499,Z 521.416,A -85,B 0,C 180,E1 -16049.053,E2 -16049.053} C_VEL
LIN {X 0,Y 305.444,Z 521.437,A -85,B 0,C 180,E1 -16051.953,E2 -16051.953} C_VEL
LIN {X 0,Y 305.459,Z 521.425,A -85,B 0,C 180,E1 -16055.114,E2 -16055.114} C_VEL
LIN {X 0,Y 305.446,Z 521.437,A -85,B 0,C 180,E1 -16058.53,E2 -16058.53} C_VEL
LIN {X 0,Y 305.457,Z 521.438,A -85,B 0,C 180,E1 -16062.588,E2 -16062.588} C_VEL
LIN {X 0,Y 305.442,Z 521.436,A -85,B 0,C 180,E1 -16066.349,E2 -16066.349} C_VEL
LIN {X 0,Y 305.457,Z 521.432,A -85,B 0,C 180,E1 -16069.893,E2 -16069.893} C_VEL
LIN {X 0,Y 305.509,Z 521.422,A -85,B 0,C 180,E1 -16074.084,E2 -16074.084} C_VEL
LIN {X 0,Y 305.514,Z 521.454,A -85,B 0,C 180,E1 -16074.39,E2 -16074.39} C_VEL
LIN {X 0,Y 309.135,Z 535.042,A -85,B 0,C 180,E1 -16077.956,E2 -16077.956} C_VEL
LIN {X 0,Y 311.949,Z 547.408,A -85,B 0,C 180,E1 -16080.971,E2 -16080.971} C_VEL
LIN {X 0,Y 312.462,Z 550.154,A -85,B 0,C 180,E1 -16081.581,E2 -16081.581} C_VEL
LIN {X 0,Y 315.592,Z 564.247,A -85,B 0,C 180,E1 -16082.229,E2 -16082.229} C_VEL
LIN {X 0,Y 319.074,Z 583.208,A -85,B 0,C 180,E1 -16083.011,E2 -16083.011} C_VEL
LIN {X 0,Y 316.971,Z 660.995,A -85,B 0,C 180,E1 -16084.779,E2 -16084.779} C_VEL
LIN {X 0,Y 316.168,Z 674.26,A -85,B 0,C 180,E1 -16085.325,E2 -16085.325} C_VEL
LIN {X 0,Y 315.262,Z 686.036,A -85,B 0,C 180,E1 -16086.065,E2 -16086.065} C_VEL
LIN {X 0,Y 314,Z 698.448,A -85,B 0,C 180,E1 -16087.115,E2 -16087.115} C_VEL
LIN {X 0,Y 312.452,Z 709.958,A -85,B 0,C 180,E1 -16088.388,E2 -16088.388} C_VEL
LIN {X 0,Y 310.836,Z 720.266,A -85,B 0,C 180,E1 -16089.831,E2 -16089.831} C_VEL
LIN {X 0,Y 309.264,Z 729.577,A -85,B 0,C 180,E1 -16091.449,E2 -16091.449} C_VEL
LIN {X 0,Y 307.901,Z 737.322,A -85,B 0,C 180,E1 -16093.114,E2 -16093.114} C_VEL
LIN {X 0,Y 306.76,Z 744.614,A -85,B 0,C 180,E1 -16095.064,E2 -16095.064} C_VEL
LIN {X 0,Y 305.477,Z 751.463,A -85,B 0,C 180,E1 -16097.376,E2 -16097.376} C_VEL
LIN {X 0,Y 304.705,Z 755.973,A -85,B 0,C 180,E1 -16099.367,E2 -16099.367} C_VEL
LIN {X 0,Y 304.376,Z 758.341,A -85,B 0,C 180,E1 -16100.699,E2 -16100.699} C_VEL
LIN {X 0,Y 303.85,Z 761.79,A -85,B 0,C 180,E1 -16103.359,E2 -16103.359} C_VEL
LIN {X 0,Y 303.708,Z 762.873,A -85,B 0,C 180,E1 -16104.689,E2 -16104.689} C_VEL
LIN {X 0,Y 303.679,Z 763.544,A -85,B 0,C 180,E1 -16106.019,E2 -16106.019} C_VEL
LIN {X 0,Y 303.637,Z 763.838,A -85,B 0,C 180,E1 -16107.347,E2 -16107.347} C_VEL
LIN {X 0,Y 303.59,Z 763.751,A -85,B 0,C 180,E1 -16108.674,E2 -16108.674} C_VEL
LIN {X 0,Y 303.609,Z 763.233,A -85,B 0,C 180,E1 -16110,E2 -16110} C_VEL
LIN {X 0,Y 303.827,Z 761.028,A -85,B 0,C 180,E1 -16112.652,E2 -16112.652} C_VEL
LIN {X 0,Y 304.188,Z 758.272,A -85,B 0,C 180,E1 -16114.638,E2 -16114.638} C_VEL
LIN {X 0,Y 304.65,Z 754.506,A -85,B 0,C 180,E1 -16116.623,E2 -16116.623} C_VEL
LIN {X 0,Y 305.301,Z 749.622,A -85,B 0,C 180,E1 -16118.605,E2 -16118.605} C_VEL
LIN {X 0,Y 306.203,Z 743.465,A -85,B 0,C 180,E1 -16120.58,E2 -16120.58} C_VEL
LIN {X 0,Y 307.417,Z 735.737,A -85,B 0,C 180,E1 -16122.543,E2 -16122.543} C_VEL
LIN {X 0,Y 308.889,Z 726.126,A -85,B 0,C 180,E1 -16124.494,E2 -16124.494} C_VEL
LIN {X 0,Y 310.304,Z 716.071,A -85,B 0,C 180,E1 -16126.107,E2 -16126.107} C_VEL
LIN {X 0,Y 311.609,Z 706.165,A -85,B 0,C 180,E1 -16127.387,E2 -16127.387} C_VEL
LIN {X 0,Y 312.836,Z 695.394,A -85,B 0,C 180,E1 -16128.501,E2 -16128.501} C_VEL
LIN {X 0,Y 313.99,Z 683.476,A -85,B 0,C 180,E1 -16129.447,E2 -16129.447} C_VEL
LIN {X 0,Y 314.791,Z 670.303,A -85,B 0,C 180,E1 -16130.203,E2 -16130.203} C_VEL
LIN {X 0,Y 315.372,Z 657.154,A -85,B 0,C 180,E1 -16130.682,E2 -16130.682} C_VEL
LIN {X 0,Y 317.078,Z 581.093,A -85,B 0,C 180,E1 -16132.399,E2 -16132.399} C_VEL
LIN {X 0,Y 312.054,Z 553.203,A -85,B 0,C 180,E1 -16133.495,E2 -16133.495} C_VEL
LIN {X 0,Y 311.426,Z 549.896,A -85,B 0,C 180,E1 -16133.657,E2 -16133.657} C_VEL
LIN {X 0,Y 311.145,Z 545.795,A -85,B 0,C 180,E1 -16134.53,E2 -16134.53} C_VEL
LIN {X 0,Y 308.712,Z 533.746,A -85,B 0,C 180,E1 -16137.394,E2 -16137.394} C_VEL
LIN {X 0,Y 305.52,Z 521.431,A -85,B 0,C 180,E1 -16140.497,E2 -16140.497} C_VEL
LIN {X 0,Y 305.465,Z 521.431,A -85,B 0,C 180,E1 -16144.077,E2 -16144.077} C_VEL
LIN {X 0,Y 305.497,Z 521.424,A -85,B 0,C 180,E1 -16146.672,E2 -16146.672} C_VEL
LIN {X 0,Y 304.828,Z 521.514,A -85,B 0,C 180,E1 -16147.771,E2 -16147.771} C_VEL
LIN {X 0,Y 301.945,Z 521.867,A -85,B 0,C 180,E1 -16149.56,E2 -16149.56} C_VEL
LIN {X 0,Y 299.514,Z 522.168,A -85,B 0,C 180,E1 -16151.011,E2 -16151.011} C_VEL
LIN {X 0,Y 298.498,Z 522.302,A -85,B 0,C 180,E1 -16152.136,E2 -16152.136} C_VEL
